LIN {X 0,Y 254.644,Z 265.777,A -85,B 0,C 180,E1 -18845.153,E2 -18845.153} C_VEL
LIN {X 0,Y 252.465,Z 261.449,A -85,B 0,C 180,E1 -18845.727,E2 -18845.727} C_VEL
LIN {X 0,Y 250.653,Z 254.367,A -85,B 0,C 180,E1 -18848.916,E2 -18848.916} C_VEL
LIN {X 0,Y 249.032,Z 248.465,A -85,B 0,C 180,E1 -18851.812,E2 -18851.812} C_VEL
LIN {X 0,Y 248.993,Z 248.471,A -85,B 0,C 180,E1 -18855.118,E2 -18855.118} C_VEL
LIN {X 0,Y 248.985,Z 248.471,A -85,B 0,C 180,E1 -18859.518,E2 -18859.518} C_VEL
LIN {X 0,Y 249.027,Z 248.458,A -85,B 0,C 180,E1 -18863.654,E2 -18863.654} C_VEL
LIN {X 0,Y 249.034,Z 248.461,A -85,B 0,C 180,E1 -18867.847,E2 -18867.847} C_VEL
LIN {X 0,Y 249.054,Z 248.454,A -85,B 0,C 180,E1 -18871.333,E2 -18871.333} C_VEL
LIN {X 0,Y 249.125,Z 248.443,A -85,B 0,C 180,E1 -18874.966,E2 -18874.966} C_VEL
LIN {X 0,Y 249.09,Z 248.448,A -85,B 0,C 180,E1 -18878.605,E2 -18878.605} C_VEL
LIN {X 0,Y 249.196,Z 248.434,A -85,B 0,C 180,E1 -18883.619,E2 -18883.619} C_VEL
LIN {X 0,Y 249.253,Z 248.426,A -85,B 0,C 180,E1 -18888.617,E2 -18888.617} C_VEL
LIN {X 0,Y 249.481,Z 248.4,A -85,B 0,C 180,E1 -18891.903,E2 -18891.903} C_VEL
LIN {X 0,Y 249.424,Z 248.409,A -85,B 0,C 180,E1 -18896.77,E2 -18896.77} C_VEL
LIN {X 0,Y 249.722,Z 248.378,A -85,B 0,C 180,E1 -18900,E2 -18900} C_VEL
LIN {X 0,Y 249.428,Z 248.403,A -85,B 0,C 180,E1 -18903.231,E2 -18903.231} C_VEL
LIN {X 0,Y 249.428,Z 248.412,A -85,B 0,C 180,E1 -18906.539,E2 -18906.539} C_VEL
LIN {X 0,Y 249.344,Z 248.42,A -85,B 0,C 180,E1 -18909.737,E2 -18909.737} C_VEL
LIN {X 0,Y 249.184,Z 248.44,A -85,B 0,C 180,E1 -18914.705,E2 -18914.705} C_VEL
LIN {X 0,Y 249.122,Z 248.44,A -85,B 0,C 180,E1 -18918.079,E2 -18918.079} C_VEL
LIN {X 0,Y 249.089,Z 248.449,A -85,B 0,C 180,E1 -18921.518,E2 -18921.518} C_VEL
LIN {X 0,Y 249.132,Z 248.446,A -85,B 0,C 180,E1 -18925.482,E2 -18925.482} C_VEL
LIN {X 0,Y 249.084,Z 248.456,A -85,B 0,C 180,E1 -18928.993,E2 -18928.993} C_VEL
LIN {X 0,Y 249.038,Z 248.463,A -85,B 0,C 180,E1 -18932.425,E2 -18932.425} C_VEL
LIN {X 0,Y 249.071,Z 248.454,A -85,B 0,C 180,E1 -18936.339,E2 -18936.339} C_VEL
LIN {X 0,Y 249.028,Z 248.466,A -85,B 0,C 180,E1 -18940.474,E2 -18940.474} C_VEL
LIN {X 0,Y 249.009,Z 248.471,A -85,B 0,C 180,E1 -18944.878,E2 -18944.878} C_VEL
LIN {X 0,Y 249.053,Z 248.62,A -85,B 0,C 180,E1 -18946.775,E2 -18946.775} C_VEL
LIN {X 0,Y 249.732,Z 251.001,A -85,B 0,C 180,E1 -18947.867,E2 -18947.867} C_VEL
LIN {X 0,Y 251.958,Z 254.871,A -85,B 0,C 180,E1 -18948.414,E2 -18948.414} C_VEL
LIN {X 0,Y 259.682,Z 268.72,A -85,B 0,C 180,E1 -18950.225,E2 -18950.225} C_VEL
LIN {X 0,Y 266.813,Z 283.218,A -85,B 0,C 180,E1 -18951.823,E2 -18951.823} C_VEL
LIN {X 0,Y 272.007,Z 295.388,A -85,B 0,C 180,E1 -18952.966,E2 -18952.966} C_VEL
LIN {X 0,Y 269.432,Z 358.338,A -85,B 0,C 180,E1 -18954.619,E2 -18954.619} C_VEL
LIN {X 0,Y 268.302,Z 371.737,A -85,B 0,C 180,E1 -18955.269,E2 -18955.269} C_VEL
LIN {X 0,Y 266.695,Z 384.328,A -85,B 0,C 180,E1 -18956.173,E2 -18956.173} C_VEL
LIN {X 0,Y 264.837,Z 395.51,A -85,B 0,C 180,E1 -18957.269,E2 -18957.269} C_VEL
LIN {X 0,Y 262.78,Z 405.83,A -85,B 0,C 180,E1 -18958.566,E2 -18958.566} C_VEL
LIN {X 0,Y 260.538,Z 415.694,A -85,B 0,C 180,E1 -18960.123,E2 -18960.123} C_VEL
LIN {X 0,Y 257.968,Z 425.167,A -85,B 0,C 180,E1 -18961.969,E2 -18961.969} C_VEL
LIN {X 0,Y 255.795,Z 433.148,A -85,B 0,C 180,E1 -18963.921,E2 -18963.921} C_VEL
LIN {X 0,Y 253.647,Z 440.407,A -85,B 0,C 180,E1 -18966.115,E2 -18966.115} C_VEL
LIN {X 0,Y 251.531,Z 447.119,A -85,B 0,C 180,E1 -18968.701,E2 -18968.701} C_VEL
LIN {X 0,Y 249.932,Z 452.023,A -85,B 0,C 180,E1 -18971.133,E2 -18971.133} C_VEL
LIN {X 0,Y 248.6,Z 456.301,A -85,B 0,C 180,E1 -18973.987,E2 -18973.987} C_VEL
LIN {X 0,Y 247.593,Z 459.227,A -85,B 0,C 180,E1 -18976.875,E2 -18976.875} C_VEL
LIN {X 0,Y 246.978,Z 460.932,A -85,B 0,C 180,E1 -18980.169,E2 -18980.169} C_VEL
LIN {X 0,Y 246.875,Z 461.202,A -85,B 0,C 180,E1 -18981.817,E2 -18981.817} C_VEL
LIN {X 0,Y 246.896,Z 461.079,A -85,B 0,C 180,E1 -18983.462,E2 -18983.462} C_VEL
LIN {X 0,Y 246.904,Z 460.527,A -85,B 0,C 180,E1 -18985.101,E2 -18985.101} C_VEL
LIN {X 0,Y 246.944,Z 459.589,A -85,B 0,C 180,E1 -18986.737,E2 -18986.737} C_VEL
LIN {X 0,Y 247.065,Z 458.263,A -85,B 0,C 180,E1 -18988.37,E2 -18988.37} C_VEL
LIN {X 0,Y 247.333,Z 455.467,A -85,B 0,C 180,E1 -18990.814,E2 -18990.814} C_VEL
LIN {X 0,Y 247.846,Z 451.66,A -85,B 0,C 180,E1 -18993.251,E2 -18993.251} C_VEL
LIN {X 0,Y 248.73,Z 446.732,A -85,B 0,C 180,E1 -18995.675,E2 -18995.675} C_VEL
LIN {X 0,Y 249.83,Z 440.548,A -85,B 0,C 180,E1 -18998.086,E2 -18998.086} C_VEL
LIN {X 0,Y 251.372,Z 432.816,A -85,B 0,C 180,E1 -19000.471,E2 -19000.471} C_VEL
LIN {X 0,Y 253.2,Z 423.156,A -85,B 0,C 180,E1 -19002.83,E2 -19002.83} C_VEL
LIN {X 0,Y 255.034,Z 413.156,A -85,B 0,C 180,E1 -19004.768,E2 -19004.768} C_VEL
LIN {X 0,Y 256.708,Z 402.883,A -85,B 0,C 180,E1 -19006.349,E2 -19006.349} C_VEL
LIN {X 0,Y 258.418,Z 390.457,A -85,B 0,C 180,E1 -19007.847,E2 -19007.847} C_VEL
LIN {X 0,Y 259.785,Z 378.325,A -85,B 0,C 180,E1 -19008.944,E2 -19008.944} C_VEL
LIN {X 0,Y 260.762,Z 365.091,A -85,B 0,C 180,E1 -19009.79,E2 -19009.79} C_VEL
LIN {X 0,Y 261.46,Z 352.137,A -85,B 0,C 180,E1 -19010.299,E2 -19010.299} C_VEL
LIN {X 0,Y 263.463,Z 286.138,A -85,B 0,C 180,E1 -19012.052,E2 -19012.052} C_VEL
LIN {X 0,Y 262.345,Z 281.579,A -85,B 0,C 180,E1 -19012.305,E2 -19012.305} C_VEL
LIN {X 0,Y 255.624,Z 264.114,A -85,B 0,C 180,E1 -19013.578,E2 -19013.578} C_VEL
LIN {X 0,Y 249.495,Z 250.179,A -85,B 0,C 180,E1 -19014.754,E2 -19014.754} C_VEL
LIN {X 0,Y 249.1,Z 248.457,A -85,B 0,C 180,E1 -19015.573,E2 -19015.573} C_VEL
LIN {X 0,Y 249.043,Z 248.465,A -85,B 0,C 180,E1 -19018.976,E2 -19018.976} C_VEL
LIN {X 0,Y 249.029,Z 248.466,A -85,B 0,C 180,E1 -19022.426,E2 -19022.426} C_VEL
LIN {X 0,Y 249.05,Z 248.462,A -85,B 0,C 180,E1 -19026.342,E2 -19026.342} C_VEL
LIN {X 0,Y 249.008,Z 248.467,A -85,B 0,C 180,E1 -19030.478,E2 -19030.478} C_VEL
LIN {X 0,Y 249.009,Z 248.468,A -85,B 0,C 180,E1 -19034.878,E2 -19034.878} C_VEL
LIN {X 0,Y 249.02,Z 248.464,A -85,B 0,C 180,E1 -19037.363,E2 -19037.363} C_VEL
LIN {X 0,Y 249.045,Z 248.46,A -85,B 0,C 180,E1 -19042.2,E2 -19042.2} C_VEL
LIN {X 0,Y 249.045,Z 248.456,A -85,B 0,C 180,E1 -19045.639,E2 -19045.639} C_VEL
LIN {X 0,Y 249.048,Z 248.454,A -85,B 0,C 180,E1 -19049.472,E2 -19049.472} C_VEL
LIN {X 0,Y 249.073,Z 248.457,A -85,B 0,C 180,E1 -19053.162,E2 -19053.162} C_VEL
LIN {X 0,Y 249.08,Z 248.438,A -85,B 0,C 180,E1 -19056.732,E2 -19056.732} C_VEL
LIN {X 0,Y 249.112,Z 248.443,A -85,B 0,C 180,E1 -19060.211,E2 -19060.211} C_VEL
LIN {X 0,Y 249.243,Z 248.434,A -85,B 0,C 180,E1 -19063.622,E2 -19063.622} C_VEL
LIN {X 0,Y 249.244,Z 248.412,A -85,B 0,C 180,E1 -19068.616,E2 -19068.616} C_VEL
LIN {X 0,Y 249.42,Z 248.405,A -85,B 0,C 180,E1 -19071.901,E2 -19071.901} C_VEL
LIN {X 0,Y 249.286,Z 248.43,A -85,B 0,C 180,E1 -19075.148,E2 -19075.148} C_VEL
LIN {X 0,Y 249.675,Z 248.377,A -85,B 0,C 180,E1 -19078.387,E2 -19078.387} C_VEL
LIN {X 0,Y 249.675,Z 248.381,A -85,B 0,C 180,E1 -19081.613,E2 -19081.613} C_VEL
LIN {X 0,Y 249.374,Z 248.413,A -85,B 0,C 180,E1 -19083.673,E2 -19083.673} C_VEL
LIN {X 0,Y 248.627,Z 248.513,A -85,B 0,C 180,E1 -19085.022,E2 -19085.022} C_VEL
LIN {X 0,Y 245.805,Z 248.865,A -85,B 0,C 180,E1 -19087.226,E2 -19087.226} C_VEL
LIN {X 0,Y 242.607,Z 249.259,A -85,B 0,C 180,E1 -19089.94,E2 -19089.94} C_VEL
LIN {X 0,Y 242.238,Z 249.299,A -85,B 0,C 180,E1 -19090.879,E2 -19090.879} C_VEL
LIN {X 0,Y 242.127,Z 249.323,A -85,B 0,C 180,E1 -19095.143,E2 -19095.143} C_VEL
LIN {X 0,Y 242.042,Z 249.326,A -85,B 0,C 180,E1 -19098.626,E2 -19098.626} C_VEL
LIN {X 0,Y 242.003,Z 249.34,A -85,B 0,C 180,E1 -19102.181,E2 -19102.181} C_VEL
LIN {X 0,Y 242.032,Z 249.33,A -85,B 0,C 180,E1 -19105.821,E2 -19105.821} C_VEL
LIN {X 0,Y 241.97,Z 249.34,A -85,B 0,C 180,E1 -19109.588,E2 -19109.588} C_VEL
LIN {X 0,Y 241.979,Z 249.341,A -85,B 0,C 180,E1 -19113.493,E2 -19113.493} C_VEL
LIN {X 0,Y 241.987,Z 249.34,A -85,B 0,C 180,E1 -19117.582,E2 -19117.582} C_VEL
LIN {X 0,Y 241.923,Z 249.348,A -85,B 0,C 180,E1 -19121.925,E2 -19121.925} C_VEL
LIN {X 0,Y 241.932,Z 249.348,A -85,B 0,C 180,E1 -19126.572,E2 -19126.572} C_VEL
LIN {X 0,Y 241.958,Z 249.344,A -85,B 0,C 180,E1 -19130.281,E2 -19130.281} C_VEL
LIN {X 0,Y 242.041,Z 249.382,A -85,B 0,C 180,E1 -19133.562,E2 -19133.562} C_VEL
LIN {X 0,Y 243.819,Z 257.168,A -85,B 0,C 180,E1 -19136.793,E2 -19136.793} C_VEL
LIN {X 0,Y 244.838,Z 261.978,A -85,B 0,C 180,E1 -19138.697,E2 -19138.697} C_VEL
LIN {X 0,Y 252.327,Z 280.988,A -85,B 0,C 180,E1 -19140.214,E2 -19140.214} C_VEL
LIN {X 0,Y 256.148,Z 308.906,A -85,B 0,C 180,E1 -19141.504,E2 -19141.504} C_VEL
LIN {X 0,Y 256.345,Z 314.755,A -85,B 0,C 180,E1 -19141.703,E2 -19141.703} C_VEL
LIN {X 0,Y 254.429,Z 371.318,A -85,B 0,C 180,E1 -19143.279,E2 -19143.279} C_VEL
LIN {X 0,Y 253.423,Z 384.264,A -85,B 0,C 180,E1 -19143.936,E2 -19143.936} C_VEL
LIN {X 0,Y 252.068,Z 396.315,A -85,B 0,C 180,E1 -19144.837,E2 -19144.837} C_VEL
LIN {X 0,Y 250.514,Z 407.691,A -85,B 0,C 180,E1 -19145.997,E2 -19145.997} C_VEL
LIN {X 0,Y 248.618,Z 419.413,A -85,B 0,C 180,E1 -19147.566,E2 -19147.566} C_VEL
LIN {X 0,Y 246.636,Z 429.94,A -85,B 0,C 180,E1 -19149.352,E2 -19149.352} C_VEL
LIN {X 0,Y 244.93,Z 439.63,A -85,B 0,C 180,E1 -19151.437,E2 -19151.437} C_VEL
LIN {X 0,Y 243.337,Z 447.877,A -85,B 0,C 180,E1 -19153.644,E2 -19153.644} C_VEL
LIN {X 0,Y 241.887,Z 455.347,A -85,B 0,C 180,E1 -19156.131,E2 -19156.131} C_VEL
LIN {X 0,Y 240.786,Z 462.227,A -85,B 0,C 180,E1 -19159.064,E2 -19159.064} C_VEL
LIN {X 0,Y 240.201,Z 466.755,A -85,B 0,C 180,E1 -19161.588,E2 -19161.588} C_VEL
LIN {X 0,Y 239.958,Z 469.138,A -85,B 0,C 180,E1 -19163.272,E2 -19163.272} C_VEL
LIN {X 0,Y 239.795,Z 471.343,A -85,B 0,C 180,E1 -19165.196,E2 -19165.196} C_VEL
LIN {X 0,Y 239.841,Z 473.685,A -85,B 0,C 180,E1 -19168.321,E2 -19168.321} C_VEL
LIN {X 0,Y 239.913,Z 474.357,A -85,B 0,C 180,E1 -19170,E2 -19170} C_VEL
LIN {X 0,Y 239.831,Z 474.635,A -85,B 0,C 180,E1 -19171.679,E2 -19171.679} C_VEL
LIN {X 0,Y 239.791,Z 474.103,A -85,B 0,C 180,E1 -19174.794,E2 -19174.794} C_VEL
LIN {X 0,Y 239.956,Z 473.052,A -85,B 0,C 180,E1 -19176.728,E2 -19176.728} C_VEL
LIN {X 0,Y 240.683,Z 470,A -85,B 0,C 180,E1 -19180.09,E2 -19180.09} C_VEL
LIN {X 0,Y 241.64,Z 466.547,A -85,B 0,C 180,E1 -19182.6,E2 -19182.6} C_VEL
LIN {X 0,Y 243.009,Z 462.026,A -85,B 0,C 180,E1 -19185.087,E2 -19185.087} C_VEL
LIN {X 0,Y 245.254,Z 455.196,A -85,B 0,C 180,E1 -19187.942,E2 -19187.942} C_VEL
LIN {X 0,Y 247.765,Z 446.972,A -85,B 0,C 180,E1 -19190.599,E2 -19190.599} C_VEL
LIN {X 0,Y 250.142,Z 438.63,A -85,B 0,C 180,E1 -19192.726,E2 -19192.726} C_VEL
LIN {X 0,Y 253.127,Z 428.044,A -85,B 0,C 180,E1 -19194.831,E2 -19194.831} C_VEL
LIN {X 0,Y 255.775,Z 417.28,A -85,B 0,C 180,E1 -19196.52,E2 -19196.52} C_VEL
LIN {X 0,Y 258.067,Z 406.797,A -85,B 0,C 180,E1 -19197.799,E2 -19197.799} C_VEL
LIN {X 0,Y 260.336,Z 394.187,A -85,B 0,C 180,E1 -19198.963,E2 -19198.963} C_VEL
LIN {X 0,Y 261.944,Z 381.626,A -85,B 0,C 180,E1 -19199.815,E2 -19199.815} C_VEL
LIN {X 0,Y 263.192,Z 368.388,A -85,B 0,C 180,E1 -19200.377,E2 -19200.377} C_VEL
LIN {X 0,Y 265.289,Z 315.913,A -85,B 0,C 180,E1 -19201.779,E2 -19201.779} C_VEL
LIN {X 0,Y 262.4,Z 297.114,A -85,B 0,C 180,E1 -19202.824,E2 -19202.824} C_VEL
LIN {X 0,Y 256.064,Z 282.546,A -85,B 0,C 180,E1 -19204.33,E2 -19204.33} C_VEL
LIN {X 0,Y 249.272,Z 269.095,A -85,B 0,C 180,E1 -19205.99,E2 -19205.99} C_VEL
LIN {X 0,Y 246.784,Z 264.532,A -85,B 0,C 180,E1 -19206.617,E2 -19206.617} C_VEL
LIN {X 0,Y 245.247,Z 261.249,A -85,B 0,C 180,E1 -19207.051,E2 -19207.051} C_VEL
LIN {X 0,Y 242.861,Z 252.644,A -85,B 0,C 180,E1 -19211.201,E2 -19211.201} C_VEL
LIN {X 0,Y 241.974,Z 249.345,A -85,B 0,C 180,E1 -19212.993,E2 -19212.993} C_VEL
LIN {X 0,Y 241.923,Z 249.351,A -85,B 0,C 180,E1 -19216.574,E2 -19216.574} C_VEL
LIN {X 0,Y 241.992,Z 249.341,A -85,B 0,C 180,E1 -19221.641,E2 -19221.641} C_VEL
LIN {X 0,Y 241.98,Z 249.341,A -85,B 0,C 180,E1 -19224.488,E2 -19224.488} C_VEL
LIN {X 0,Y 241.954,Z 249.345,A -85,B 0,C 180,E1 -19228.477,E2 -19228.477} C_VEL
LIN {X 0,Y 241.973,Z 249.343,A -85,B 0,C 180,E1 -19232.308,E2 -19232.308} C_VEL
LIN {X 0,Y 242.035,Z 249.335,A -85,B 0,C 180,E1 -19236.014,E2 -19236.014} C_VEL
LIN {X 0,Y 242.022,Z 249.33,A -85,B 0,C 180,E1 -19239.607,E2 -19239.607} C_VEL
LIN {X 0,Y 242.116,Z 249.316,A -85,B 0,C 180,E1 -19243.316,E2 -19243.316} C_VEL
LIN {X 0,Y 242.185,Z 249.305,A -85,B 0,C 180,E1 -19248.28,E2 -19248.28} C_VEL
LIN {X 0,Y 242.428,Z 249.28,A -85,B 0,C 180,E1 -19251.666,E2 -19251.666} C_VEL
LIN {X 0,Y 242.248,Z 249.306,A -85,B 0,C 180,E1 -19255.007,E2 -19255.007} C_VEL
LIN {X 0,Y 242.632,Z 249.248,A -85,B 0,C 180,E1 -19258.34,E2 -19258.34} C_VEL
LIN {X 0,Y 242.634,Z 249.256,A -85,B 0,C 180,E1 -19261.66,E2 -19261.66} C_VEL
LIN {X 0,Y 242.402,Z 249.289,A -85,B 0,C 180,E1 -19266.66,E2 -19266.66} C_VEL
LIN {X 0,Y 242.267,Z 249.305,A -85,B 0,C 180,E1 -19270.024,E2 -19270.024} C_VEL
LIN {X 0,Y 242.14,Z 249.319,A -85,B 0,C 180,E1 -19275.143,E2 -19275.143} C_VEL
LIN {X 0,Y 242.062,Z 249.32,A -85,B 0,C 180,E1 -19278.625,E2 -19278.625} C_VEL
LIN {X 0,Y 242.014,Z 249.326,A -85,B 0,C 180,E1 -19282.18,E2 -19282.18} C_VEL
LIN {X 0,Y 242.068,Z 249.323,A -85,B 0,C 180,E1 -19285.838,E2 -19285.838} C_VEL
LIN {X 0,Y 242.032,Z 249.33,A -85,B 0,C 180,E1 -19289.58,E2 -19289.58} C_VEL
LIN {X 0,Y 241.993,Z 249.336,A -85,B 0,C 180,E1 -19293.491,E2 -19293.491} C_VEL
LIN {X 0,Y 242.004,Z 249.341,A -85,B 0,C 180,E1 -19297.58,E2 -19297.58} C_VEL
LIN {X 0,Y 241.946,Z 249.345,A -85,B 0,C 180,E1 -19301.921,E2 -19301.921} C_VEL
LIN {X 0,Y 241.989,Z 249.526,A -85,B 0,C 180,E1 -19305.666,E2 -19305.666} C_VEL
LIN {X 0,Y 242.518,Z 251.239,A -85,B 0,C 180,E1 -19306.48,E2 -19306.48} C_VEL
LIN {X 0,Y 244.824,Z 255.198,A -85,B 0,C 180,E1 -19307.087,E2 -19307.087} C_VEL
LIN {X 0,Y 252.458,Z 268.434,A -85,B 0,C 180,E1 -19308.985,E2 -19308.985} C_VEL
LIN {X 0,Y 259.973,Z 283.303,A -85,B 0,C 180,E1 -19310.763,E2 -19310.763} C_VEL
LIN {X 0,Y 266.007,Z 297.202,A -85,B 0,C 180,E1 -19312.153,E2 -19312.153} C_VEL
LIN {X 0,Y 263.489,Z 358.084,A -85,B 0,C 180,E1 -19313.784,E2 -19313.784} C_VEL
LIN {X 0,Y 262.384,Z 371.255,A -85,B 0,C 180,E1 -19314.427,E2 -19314.427} C_VEL
LIN {X 0,Y 260.789,Z 383.471,A -85,B 0,C 180,E1 -19315.299,E2 -19315.299} C_VEL
LIN {X 0,Y 258.862,Z 394.95,A -85,B 0,C 180,E1 -19316.415,E2 -19316.415} C_VEL
LIN {X 0,Y 256.658,Z 405.402,A -85,B 0,C 180,E1 -19317.726,E2 -19317.726} C_VEL
LIN {X 0,Y 254.213,Z 415.793,A -85,B 0,C 180,E1 -19319.389,E2 -19319.389} C_VEL
LIN {X 0,Y 251.641,Z 424.936,A -85,B 0,C 180,E1 -19321.199,E2 -19321.199} C_VEL
LIN {X 0,Y 249.326,Z 432.987,A -85,B 0,C 180,E1 -19323.192,E2 -19323.192} C_VEL
LIN {X 0,Y 246.916,Z 440.834,A -85,B 0,C 180,E1 -19325.62,E2 -19325.62} C_VEL
LIN {X 0,Y 244.835,Z 447.097,A -85,B 0,C 180,E1 -19328.089,E2 -19328.089} C_VEL
LIN {X 0,Y 243.12,Z 452.049,A -85,B 0,C 180,E1 -19330.583,E2 -19330.583} C_VEL
LIN {X 0,Y 241.866,Z 455.855,A -85,B 0,C 180,E1 -19333.108,E2 -19333.108} C_VEL
LIN {X 0,Y 241.182,Z 457.808,A -85,B 0,C 180,E1 -19334.796,E2 -19334.796} C_VEL
LIN {X 0,Y 240.616,Z 459.344,A -85,B 0,C 180,E1 -19336.487,E2 -19336.487} C_VEL
LIN {X 0,Y 240.153,Z 460.428,A -85,B 0,C 180,E1 -19338.179,E2 -19338.179} C_VEL
LIN {X 0,Y 239.798,Z 461.39,A -85,B 0,C 180,E1 -19341.573,E2 -19341.573} C_VEL
LIN {X 0,Y 239.788,Z 461.294,A -85,B 0,C 180,E1 -19343.267,E2 -19343.267} C_VEL
LIN {X 0,Y 239.804,Z 460.669,A -85,B 0,C 180,E1 -19345.173,E2 -19345.173} C_VEL
LIN {X 0,Y 239.966,Z 458.546,A -85,B 0,C 180,E1 -19348.322,E2 -19348.322} C_VEL
LIN {X 0,Y 240.248,Z 455.79,A -85,B 0,C 180,E1 -19350.838,E2 -19350.838} C_VEL
LIN {X 0,Y 240.771,Z 452.026,A -85,B 0,C 180,E1 -19353.347,E2 -19353.347} C_VEL
LIN {X 0,Y 241.675,Z 447.145,A -85,B 0,C 180,E1 -19355.842,E2 -19355.842} C_VEL
LIN {X 0,Y 242.82,Z 441.011,A -85,B 0,C 180,E1 -19358.321,E2 -19358.321} C_VEL
LIN {X 0,Y 244.417,Z 433.366,A -85,B 0,C 180,E1 -19360.772,E2 -19360.772} C_VEL
LIN {X 0,Y 246.316,Z 423.776,A -85,B 0,C 180,E1 -19363.195,E2 -19363.195} C_VEL
LIN {X 0,Y 248.217,Z 413.88,A -85,B 0,C 180,E1 -19365.183,E2 -19365.183} C_VEL
LIN {X 0,Y 250.058,Z 403.078,A -85,B 0,C 180,E1 -19366.897,E2 -19366.897} C_VEL
LIN {X 0,Y 251.639,Z 392.119,A -85,B 0,C 180,E1 -19368.27,E2 -19368.27} C_VEL
LIN {X 0,Y 253.115,Z 379.659,A -85,B 0,C 180,E1 -19369.463,E2 -19369.463} C_VEL
LIN {X 0,Y 254.184,Z 367.02,A -85,B 0,C 180,E1 -19370.325,E2 -19370.325} C_VEL
LIN {X 0,Y 254.817,Z 355.22,A -85,B 0,C 180,E1 -19370.852,E2 -19370.852} C_VEL
LIN {X 0,Y 257.05,Z 287.162,A -85,B 0,C 180,E1 -19372.709,E2 -19372.709} C_VEL
LIN {X 0,Y 255.55,Z 282.213,A -85,B 0,C 180,E1 -19373.027,E2 -19373.027} C_VEL
LIN {X 0,Y 249.926,Z 267.53,A -85,B 0,C 180,E1 -19374.141,E2 -19374.141} C_VEL
LIN {X 0,Y 242.234,Z 250.331,A -85,B 0,C 180,E1 -19375.704,E2 -19375.704} C_VEL
LIN {X 0,Y 242.011,Z 249.341,A -85,B 0,C 180,E1 -19376.24,E2 -19376.24} C_VEL
LIN {X 0,Y 241.972,Z 249.343,A -85,B 0,C 180,E1 -19379.588,E2 -19379.588} C_VEL
LIN {X 0,Y 241.981,Z 249.342,A -85,B 0,C 180,E1 -19383.492,E2 -19383.492} C_VEL
LIN {X 0,Y 241.991,Z 249.34,A -85,B 0,C 180,E1 -19387.581,E2 -19387.581} C_VEL
LIN {X 0,Y 241.94,Z 249.345,A -85,B 0,C 180,E1 -19391.922,E2 -19391.922} C_VEL
LIN {X 0,Y 241.938,Z 249.349,A -85,B 0,C 180,E1 -19396.57,E2 -19396.57} C_VEL
LIN {X 0,Y 241.958,Z 249.346,A -85,B 0,C 180,E1 -19400.281,E2 -19400.281} C_VEL
LIN {X 0,Y 241.989,Z 249.341,A -85,B 0,C 180,E1 -19404.489,E2 -19404.489} C_VEL
LIN {X 0,Y 241.974,Z 249.325,A -85,B 0,C 180,E1 -19408.479,E2 -19408.479} C_VEL
LIN {X 0,Y 242.004,Z 249.339,A -85,B 0,C 180,E1 -19412.312,E2 -19412.312} C_VEL
LIN {X 0,Y 242.058,Z 249.319,A -85,B 0,C 180,E1 -19416.016,E2 -19416.016} C_VEL
LIN {X 0,Y 242.039,Z 249.322,A -85,B 0,C 180,E1 -19419.608,E2 -19419.608} C_VEL
LIN {X 0,Y 242.164,Z 249.316,A -85,B 0,C 180,E1 -19423.278,E2 -19423.278} C_VEL
LIN {X 0,Y 242.181,Z 249.292,A -85,B 0,C 180,E1 -19428.279,E2 -19428.279} C_VEL
LIN {X 0,Y 242.373,Z 249.282,A -85,B 0,C 180,E1 -19431.663,E2 -19431.663} C_VEL
LIN {X 0,Y 242.246,Z 249.307,A -85,B 0,C 180,E1 -19435.007,E2 -19435.007} C_VEL
LIN {X 0,Y 242.635,Z 249.253,A -85,B 0,C 180,E1 -19438.34,E2 -19438.34} C_VEL
LIN {X 0,Y 242.635,Z 249.258,A -85,B 0,C 180,E1 -19441.66,E2 -19441.66} C_VEL
LIN {X 0,Y 242.434,Z 249.288,A -85,B 0,C 180,E1 -19446.659,E2 -19446.659} C_VEL
LIN {X 0,Y 242.346,Z 249.291,A -85,B 0,C 180,E1 -19450.02,E2 -19450.02} C_VEL
LIN {X 0,Y 242.238,Z 249.299,A -85,B 0,C 180,E1 -19450.879,E2 -19450.879} C_VEL
LIN {X 0,Y 241.474,Z 249.397,A -85,B 0,C 180,E1 -19452.266,E2 -19452.266} C_VEL
LIN {X 0,Y 238.548,Z 249.771,A -85,B 0,C 180,E1 -19454.528,E2 -19454.528} C_VEL
LIN {X 0,Y 236.108,Z 250.073,A -85,B 0,C 180,E1 -19456.371,E2 -19456.371} C_VEL
LIN {X 0,Y 235.061,Z 250.197,A -85,B 0,C 180,E1 -19457.802,E2 -19457.802} C_VEL
LIN {X 0,Y 234.971,Z 250.205,A -85,B 0,C 180,E1 -19458.287,E2 -19458.287} C_VEL
LIN {X 0,Y 234.986,Z 250.213,A -85,B 0,C 180,E1 -19462.005,E2 -19462.005} C_VEL
LIN {X 0,Y 234.946,Z 250.217,A -85,B 0,C 180,E1 -19466.66,E2 -19466.66} C_VEL
LIN {X 0,Y 234.899,Z 250.22,A -85,B 0,C 180,E1 -19470.572,E2 -19470.572} C_VEL
LIN {X 0,Y 234.93,Z 250.217,A -85,B 0,C 180,E1 -19474.638,E2 -19474.638} C_VEL
LIN {X 0,Y 234.911,Z 250.22,A -85,B 0,C 180,E1 -19478.935,E2 -19478.935} C_VEL
LIN {X 0,Y 234.876,Z 250.227,A -85,B 0,C 180,E1 -19483.489,E2 -19483.489} C_VEL
LIN {X 0,Y 234.885,Z 250.226,A -85,B 0,C 180,E1 -19486.514,E2 -19486.514} C_VEL
LIN {X 0,Y 234.922,Z 250.22,A -85,B 0,C 180,E1 -19491.079,E2 -19491.079} C_VEL
LIN {X 0,Y 234.991,Z 250.273,A -85,B 0,C 180,E1 -19492.861,E2 -19492.861} C_VEL
LIN {X 0,Y 237.052,Z 259.31,A -85,B 0,C 180,E1 -19496.738,E2 -19496.738} C_VEL
LIN {X 0,Y 237.647,Z 261.991,A -85,B 0,C 180,E1 -19497.753,E2 -19497.753} C_VEL
LIN {X 0,Y 244.944,Z 279.897,A -85,B 0,C 180,E1 -19499.295,E2 -19499.295} C_VEL
LIN {X 0,Y 246.394,Z 284.268,A -85,B 0,C 180,E1 -19499.615,E2 -19499.615} C_VEL
LIN {X 0,Y 249.991,Z 311.683,A -85,B 0,C 180,E1 -19500.91,E2 -19500.91} C_VEL
LIN {X 0,Y 247.972,Z 371.131,A -85,B 0,C 180,E1 -19502.609,E2 -19502.609} C_VEL
LIN {X 0,Y 246.883,Z 384.479,A -85,B 0,C 180,E1 -19503.305,E2 -19503.305} C_VEL
LIN {X 0,Y 245.4,Z 397.49,A -85,B 0,C 180,E1 -19504.331,E2 -19504.331} C_VEL
LIN {X 0,Y 243.497,Z 410.101,A -85,B 0,C 180,E1 -19505.714,E2 -19505.714} C_VEL
LIN {X 0,Y 241.552,Z 421.344,A -85,B 0,C 180,E1 -19507.325,E2 -19507.325} C_VEL
LIN {X 0,Y 239.755,Z 430.429,A -85,B 0,C 180,E1 -19508.956,E2 -19508.956} C_VEL
LIN {X 0,Y 238.016,Z 439.757,A -85,B 0,C 180,E1 -19511.047,E2 -19511.047} C_VEL
LIN {X 0,Y 236.482,Z 447.434,A -85,B 0,C 180,E1 -19513.157,E2 -19513.157} C_VEL
LIN {X 0,Y 234.978,Z 454.949,A -85,B 0,C 180,E1 -19515.715,E2 -19515.715} C_VEL
LIN {X 0,Y 233.775,Z 461.881,A -85,B 0,C 180,E1 -19518.731,E2 -19518.731} C_VEL
LIN {X 0,Y 233.142,Z 466.445,A -85,B 0,C 180,E1 -19521.331,E2 -19521.331} C_VEL
LIN {X 0,Y 232.891,Z 468.845,A -85,B 0,C 180,E1 -19523.067,E2 -19523.067} C_VEL
LIN {X 0,Y 232.714,Z 471.294,A -85,B 0,C 180,E1 -19525.278,E2 -19525.278} C_VEL
LIN {X 0,Y 232.752,Z 473.453,A -85,B 0,C 180,E1 -19528.27,E2 -19528.27} C_VEL
LIN {X 0,Y 232.823,Z 474.139,A -85,B 0,C 180,E1 -19530,E2 -19530} C_VEL
LIN {X 0,Y 232.743,Z 474.431,A -85,B 0,C 180,E1 -19531.73,E2 -19531.73} C_VEL
LIN {X 0,Y 232.707,Z 474.006,A -85,B 0,C 180,E1 -19534.702,E2 -19534.702} C_VEL
LIN {X 0,Y 232.894,Z 472.905,A -85,B 0,C 180,E1 -19536.933,E2 -19536.933} C_VEL
LIN {X 0,Y 233.681,Z 469.887,A -85,B 0,C 180,E1 -19540.396,E2 -19540.396} C_VEL
LIN {X 0,Y 234.672,Z 466.462,A -85,B 0,C 180,E1 -19542.98,E2 -19542.98} C_VEL
LIN {X 0,Y 236.157,Z 461.976,A -85,B 0,C 180,E1 -19545.536,E2 -19545.536} C_VEL
LIN {X 0,Y 238.474,Z 455.203,A -85,B 0,C 180,E1 -19548.47,E2 -19548.47} C_VEL
LIN {X 0,Y 240.92,Z 447.621,A -85,B 0,C 180,E1 -19551.015,E2 -19551.015} C_VEL
LIN {X 0,Y 243.601,Z 438.752,A -85,B 0,C 180,E1 -19553.372,E2 -19553.372} C_VEL
LIN {X 0,Y 246.727,Z 428.238,A -85,B 0,C 180,E1 -19555.521,E2 -19555.521} C_VEL
LIN {X 0,Y 249.454,Z 417.558,A -85,B 0,C 180,E1 -19557.247,E2 -19557.247} C_VEL
LIN {X 0,Y 251.835,Z 407.215,A -85,B 0,C 180,E1 -19558.549,E2 -19558.549} C_VEL
LIN {X 0,Y 254.18,Z 394.816,A -85,B 0,C 180,E1 -19559.734,E2 -19559.734} C_VEL
LIN {X 0,Y 255.931,Z 381.785,A -85,B 0,C 180,E1 -19560.646,E2 -19560.646} C_VEL
LIN {X 0,Y 257.233,Z 368.889,A -85,B 0,C 180,E1 -19561.215,E2 -19561.215} C_VEL
LIN {X 0,Y 259.356,Z 315.813,A -85,B 0,C 180,E1 -19562.677,E2 -19562.677} C_VEL
LIN {X 0,Y 256.73,Z 299.566,A -85,B 0,C 180,E1 -19563.639,E2 -19563.639} C_VEL
LIN {X 0,Y 250.701,Z 285.754,A -85,B 0,C 180,E1 -19565.138,E2 -19565.138} C_VEL
LIN {X 0,Y 244.162,Z 272.639,A -85,B 0,C 180,E1 -19566.816,E2 -19566.816} C_VEL
LIN {X 0,Y 239.939,Z 264.906,A -85,B 0,C 180,E1 -19567.944,E2 -19567.944} C_VEL
LIN {X 0,Y 237.882,Z 260.913,A -85,B 0,C 180,E1 -19568.571,E2 -19568.571} C_VEL
LIN {X 0,Y 235.596,Z 252.632,A -85,B 0,C 180,E1 -19572.801,E2 -19572.801} C_VEL
LIN {X 0,Y 234.903,Z 250.226,A -85,B 0,C 180,E1 -19574.196,E2 -19574.196} C_VEL
LIN {X 0,Y 234.865,Z 250.229,A -85,B 0,C 180,E1 -19578.828,E2 -19578.828} C_VEL
LIN {X 0,Y 234.918,Z 250.222,A -85,B 0,C 180,E1 -19581.079,E2 -19581.079} C_VEL
LIN {X 0,Y 234.926,Z 250.218,A -85,B 0,C 180,E1 -19585.361,E2 -19585.361} C_VEL
LIN {X 0,Y 234.9,Z 250.219,A -85,B 0,C 180,E1 -19589.428,E2 -19589.428} C_VEL
LIN {X 0,Y 234.97,Z 250.208,A -85,B 0,C 180,E1 -19593.806,E2 -19593.806} C_VEL
LIN {X 0,Y 234.991,Z 250.203,A -85,B 0,C 180,E1 -19598.968,E2 -19598.968} C_VEL
LIN {X 0,Y 235.057,Z 250.195,A -85,B 0,C 180,E1 -19603.092,E2 -19603.092} C_VEL
LIN {X 0,Y 235.116,Z 250.185,A -85,B 0,C 180,E1 -19607.922,E2 -19607.922} C_VEL
LIN {X 0,Y 235.377,Z 250.16,A -85,B 0,C 180,E1 -19611.414,E2 -19611.414} C_VEL
LIN {X 0,Y 235.403,Z 250.149,A -85,B 0,C 180,E1 -19613.141,E2 -19613.141} C_VEL
LIN {X 0,Y 235.592,Z 250.124,A -85,B 0,C 180,E1 -19618.291,E2 -19618.291} C_VEL
LIN {X 0,Y 235.594,Z 250.132,A -85,B 0,C 180,E1 -19621.71,E2 -19621.71} C_VEL
LIN {X 0,Y 235.353,Z 250.164,A -85,B 0,C 180,E1 -19626.86,E2 -19626.86} C_VEL
LIN {X 0,Y 235.213,Z 250.185,A -85,B 0,C 180,E1 -19630.328,E2 -19630.328} C_VEL
LIN {X 0,Y 235.095,Z 250.201,A -85,B 0,C 180,E1 -19635.608,E2 -19635.608} C_VEL
LIN {X 0,Y 235.002,Z 250.203,A -85,B 0,C 180,E1 -19639.206,E2 -19639.206} C_VEL
LIN {X 0,Y 234.963,Z 250.204,A -85,B 0,C 180,E1 -19642.883,E2 -19642.883} C_VEL
LIN {X 0,Y 234.971,Z 250.205,A -85,B 0,C 180,E1 -19646.657,E2 -19646.657} C_VEL
LIN {X 0,Y 234.934,Z 250.214,A -85,B 0,C 180,E1 -19650.568,E2 -19650.568} C_VEL
LIN {X 0,Y 234.962,Z 250.217,A -85,B 0,C 180,E1 -19654.633,E2 -19654.633} C_VEL
LIN {X 0,Y 234.943,Z 250.215,A -85,B 0,C 180,E1 -19658.945,E2 -19658.945} C_VEL
LIN {X 0,Y 234.892,Z 250.225,A -85,B 0,C 180,E1 -19663.485,E2 -19663.485} C_VEL
LIN {X 0,Y 234.921,Z 250.371,A -85,B 0,C 180,E1 -19664.434,E2 -19664.434} C_VEL
LIN {X 0,Y 235.231,Z 251.484,A -85,B 0,C 180,E1 -19664.96,E2 -19664.96} C_VEL
LIN {X 0,Y 236.986,Z 254.584,A -85,B 0,C 180,E1 -19665.464,E2 -19665.464} C_VEL
LIN {X 0,Y 238.679,Z 257.151,A -85,B 0,C 180,E1 -19665.922,E2 -19665.922} C_VEL
LIN {X 0,Y 246.235,Z 270.09,A -85,B 0,C 180,E1 -19667.91,E2 -19667.91} C_VEL
LIN {X 0,Y 253.137,Z 283.463,A -85,B 0,C 180,E1 -19669.632,E2 -19669.632} C_VEL
LIN {X 0,Y 259.557,Z 297.842,A -85,B 0,C 180,E1 -19671.183,E2 -19671.183} C_VEL
LIN {X 0,Y 260.183,Z 299.383,A -85,B 0,C 180,E1 -19671.333,E2 -19671.333} C_VEL
LIN {X 0,Y 257.512,Z 358.954,A -85,B 0,C 180,E1 -19672.956,E2 -19672.956} C_VEL
LIN {X 0,Y 256.311,Z 372.305,A -85,B 0,C 180,E1 -19673.633,E2 -19673.633} C_VEL
LIN {X 0,Y 254.576,Z 384.84,A -85,B 0,C 180,E1 -19674.568,E2 -19674.568} C_VEL
LIN {X 0,Y 252.577,Z 395.993,A -85,B 0,C 180,E1 -19675.705,E2 -19675.705} C_VEL
LIN {X 0,Y 250.317,Z 406.287,A -85,B 0,C 180,E1 -19677.045,E2 -19677.045} C_VEL
LIN {X 0,Y 247.955,Z 415.848,A -85,B 0,C 180,E1 -19678.611,E2 -19678.611} C_VEL
LIN {X 0,Y 245.376,Z 424.709,A -85,B 0,C 180,E1 -19680.391,E2 -19680.391} C_VEL
LIN {X 0,Y 242.909,Z 432.83,A -85,B 0,C 180,E1 -19682.424,E2 -19682.424} C_VEL
LIN {X 0,Y 240.434,Z 440.508,A -85,B 0,C 180,E1 -19684.82,E2 -19684.82} C_VEL
LIN {X 0,Y 238.173,Z 447.08,A -85,B 0,C 180,E1 -19687.443,E2 -19687.443} C_VEL
LIN {X 0,Y 236.349,Z 452.077,A -85,B 0,C 180,E1 -19690.004,E2 -19690.004} C_VEL
LIN {X 0,Y 234.985,Z 455.926,A -85,B 0,C 180,E1 -19692.597,E2 -19692.597} C_VEL
LIN {X 0,Y 234.259,Z 457.899,A -85,B 0,C 180,E1 -19694.335,E2 -19694.335} C_VEL
LIN {X 0,Y 233.637,Z 459.455,A -85,B 0,C 180,E1 -19696.075,E2 -19696.075} C_VEL
LIN {X 0,Y 233.135,Z 460.578,A -85,B 0,C 180,E1 -19697.818,E2 -19697.818} C_VEL
LIN {X 0,Y 232.707,Z 461.578,A -85,B 0,C 180,E1 -19701.315,E2 -19701.315} C_VEL
LIN {X 0,Y 232.694,Z 461.502,A -85,B 0,C 180,E1 -19703.061,E2 -19703.061} C_VEL
LIN {X 0,Y 232.715,Z 460.795,A -85,B 0,C 180,E1 -19705.281,E2 -19705.281} C_VEL
LIN {X 0,Y 232.869,Z 458.83,A -85,B 0,C 180,E1 -19708.27,E2 -19708.27} C_VEL
LIN {X 0,Y 233.166,Z 456.113,A -85,B 0,C 180,E1 -19710.863,E2 -19710.863} C_VEL
LIN {X 0,Y 233.699,Z 452.392,A -85,B 0,C 180,E1 -19713.448,E2 -19713.448} C_VEL
LIN {X 0,Y 234.625,Z 447.557,A -85,B 0,C 180,E1 -19716.018,E2 -19716.018} C_VEL
LIN {X 0,Y 235.816,Z 441.472,A -85,B 0,C 180,E1 -19718.57,E2 -19718.57} C_VEL
LIN {X 0,Y 237.47,Z 433.904,A -85,B 0,C 180,E1 -19721.091,E2 -19721.091} C_VEL
LIN {X 0,Y 239.444,Z 424.393,A -85,B 0,C 180,E1 -19723.58,E2 -19723.58} C_VEL
LIN {X 0,Y 241.415,Z 414.581,A -85,B 0,C 180,E1 -19725.622,E2 -19725.622} C_VEL
LIN {X 0,Y 243.374,Z 403.65,A -85,B 0,C 180,E1 -19727.421,E2 -19727.421} C_VEL
LIN {X 0,Y 245.142,Z 391.721,A -85,B 0,C 180,E1 -19728.948,E2 -19728.948} C_VEL
LIN {X 0,Y 246.608,Z 379.792,A -85,B 0,C 180,E1 -19730.106,E2 -19730.106} C_VEL
LIN {X 0,Y 247.702,Z 367.119,A -85,B 0,C 180,E1 -19730.99,E2 -19730.99} C_VEL
LIN {X 0,Y 248.48,Z 353.741,A -85,B 0,C 180,E1 -19731.573,E2 -19731.573} C_VEL
LIN {X 0,Y 250.735,Z 288.342,A -85,B 0,C 180,E1 -19733.386,E2 -19733.386} C_VEL
LIN {X 0,Y 244.746,Z 272.181,A -85,B 0,C 180,E1 -19734.627,E2 -19734.627} C_VEL
LIN {X 0,Y 236.762,Z 254.246,A -85,B 0,C 180,E1 -19736.28,E2 -19736.28} C_VEL
LIN {X 0,Y 235.162,Z 251.18,A -85,B 0,C 180,E1 -19736.609,E2 -19736.609} C_VEL
LIN {X 0,Y 235.025,Z 250.631,A -85,B 0,C 180,E1 -19736.65,E2 -19736.65} C_VEL
LIN {X 0,Y 234.959,Z 250.219,A -85,B 0,C 180,E1 -19736.899,E2 -19736.899} C_VEL
LIN {X 0,Y 234.901,Z 250.226,A -85,B 0,C 180,E1 -19740.572,E2 -19740.572} C_VEL
LIN {X 0,Y 234.932,Z 250.221,A -85,B 0,C 180,E1 -19744.638,E2 -19744.638} C_VEL
LIN {X 0,Y 234.943,Z 250.219,A -85,B 0,C 180,E1 -19748.944,E2 -19748.944} C_VEL
LIN {X 0,Y 234.891,Z 250.224,A -85,B 0,C 180,E1 -19753.485,E2 -19753.485} C_VEL
LIN {X 0,Y 234.891,Z 250.226,A -85,B 0,C 180,E1 -19756.514,E2 -19756.514} C_VEL
LIN {X 0,Y 234.919,Z 250.219,A -85,B 0,C 180,E1 -19761.078,E2 -19761.078} C_VEL
LIN {X 0,Y 234.932,Z 250.214,A -85,B 0,C 180,E1 -19765.362,E2 -19765.362} C_VEL
LIN {X 0,Y 234.923,Z 250.213,A -85,B 0,C 180,E1 -19769.431,E2 -19769.431} C_VEL
LIN {X 0,Y 234.995,Z 250.21,A -85,B 0,C 180,E1 -19773.794,E2 -19773.794} C_VEL
LIN {X 0,Y 235.013,Z 250.19,A -85,B 0,C 180,E1 -19778.97,E2 -19778.97} C_VEL
LIN {X 0,Y 235.098,Z 250.197,A -85,B 0,C 180,E1 -19783.059,E2 -19783.059} C_VEL
LIN {X 0,Y 235.115,Z 250.172,A -85,B 0,C 180,E1 -19787.922,E2 -19787.922} C_VEL
LIN {X 0,Y 235.313,Z 250.161,A -85,B 0,C 180,E1 -19791.412,E2 -19791.412} C_VEL
LIN {X 0,Y 235.206,Z 250.185,A -85,B 0,C 180,E1 -19794.857,E2 -19794.857} C_VEL
LIN {X 0,Y 235.595,Z 250.13,A -85,B 0,C 180,E1 -19798.29,E2 -19798.29} C_VEL
LIN {X 0,Y 235.595,Z 250.135,A -85,B 0,C 180,E1 -19801.709,E2 -19801.709} C_VEL
LIN {X 0,Y 235.406,Z 250.163,A -85,B 0,C 180,E1 -19806.858,E2 -19806.858} C_VEL
LIN {X 0,Y 235.254,Z 250.171,A -85,B 0,C 180,E1 -19810.326,E2 -19810.326} C_VEL
LIN {X 0,Y 235.075,Z 250.201,A -85,B 0,C 180,E1 -19815.609,E2 -19815.609} C_VEL
LIN {X 0,Y 234.971,Z 250.205,A -85,B 0,C 180,E1 -19818.287,E2 -19818.287} C_VEL
LIN {X 0,Y 234.288,Z 250.294,A -85,B 0,C 180,E1 -19819.717,E2 -19819.717} C_VEL
LIN {X 0,Y 231.422,Z 250.657,A -85,B 0,C 180,E1 -19822.051,E2 -19822.051} C_VEL
LIN {X 0,Y 229.002,Z 250.956,A -85,B 0,C 180,E1 -19823.954,E2 -19823.954} C_VEL
LIN {X 0,Y 227.978,Z 251.08,A -85,B 0,C 180,E1 -19825.431,E2 -19825.431} C_VEL
LIN {X 0,Y 227.901,Z 251.09,A -85,B 0,C 180,E1 -19825.932,E2 -19825.932} C_VEL
LIN {X 0,Y 227.874,Z 251.094,A -85,B 0,C 180,E1 -19830.281,E2 -19830.281} C_VEL
LIN {X 0,Y 227.877,Z 251.098,A -85,B 0,C 180,E1 -19833.72,E2 -19833.72} C_VEL
LIN {X 0,Y 227.843,Z 251.103,A -85,B 0,C 180,E1 -19838.091,E2 -19838.091} C_VEL
LIN {X 0,Y 227.801,Z 251.108,A -85,B 0,C 180,E1 -19842.745,E2 -19842.745} C_VEL
LIN {X 0,Y 227.81,Z 251.103,A -85,B 0,C 180,E1 -19847.257,E2 -19847.257} C_VEL
LIN {X 0,Y 227.948,Z 251.157,A -85,B 0,C 180,E1 -19852.108,E2 -19852.108} C_VEL
LIN {X 0,Y 229.811,Z 259.073,A -85,B 0,C 180,E1 -19855.66,E2 -19855.66} C_VEL
LIN {X 0,Y 230.312,Z 261.449,A -85,B 0,C 180,E1 -19856.683,E2 -19856.683} C_VEL
LIN {X 0,Y 238.618,Z 281.491,A -85,B 0,C 180,E1 -19858.542,E2 -19858.542} C_VEL
LIN {X 0,Y 240.257,Z 286.288,A -85,B 0,C 180,E1 -19858.915,E2 -19858.915} C_VEL
LIN {X 0,Y 243.634,Z 312.541,A -85,B 0,C 180,E1 -19860.197,E2 -19860.197} C_VEL
LIN {X 0,Y 241.565,Z 370.802,A -85,B 0,C 180,E1 -19861.899,E2 -19861.899} C_VEL
LIN {X 0,Y 240.453,Z 383.921,A -85,B 0,C 180,E1 -19862.591,E2 -19862.591} C_VEL
LIN {X 0,Y 238.972,Z 396.528,A -85,B 0,C 180,E1 -19863.588,E2 -19863.588} C_VEL
LIN {X 0,Y 237.294,Z 407.729,A -85,B 0,C 180,E1 -19864.802,E2 -19864.802} C_VEL
LIN {X 0,Y 235.264,Z 419.373,A -85,B 0,C 180,E1 -19866.45,E2 -19866.45} C_VEL
LIN {X 0,Y 233.055,Z 429.834,A -85,B 0,C 180,E1 -19868.321,E2 -19868.321} C_VEL
LIN {X 0,Y 231.222,Z 439.255,A -85,B 0,C 180,E1 -19870.467,E2 -19870.467} C_VEL
LIN {X 0,Y 230.017,Z 445.555,A -85,B 0,C 180,E1 -19872.209,E2 -19872.209} C_VEL
LIN {X 0,Y 228.312,Z 453.42,A -85,B 0,C 180,E1 -19874.832,E2 -19874.832} C_VEL
LIN {X 0,Y 227.035,Z 459.702,A -85,B 0,C 180,E1 -19877.485,E2 -19877.485} C_VEL
LIN {X 0,Y 226.279,Z 464.699,A -85,B 0,C 180,E1 -19880.164,E2 -19880.164} C_VEL
LIN {X 0,Y 225.821,Z 468.551,A -85,B 0,C 180,E1 -19882.849,E2 -19882.849} C_VEL
LIN {X 0,Y 225.625,Z 471.251,A -85,B 0,C 180,E1 -19885.393,E2 -19885.393} C_VEL
LIN {X 0,Y 225.666,Z 473.22,A -85,B 0,C 180,E1 -19888.215,E2 -19888.215} C_VEL
LIN {X 0,Y 225.734,Z 473.921,A -85,B 0,C 180,E1 -19890,E2 -19890} C_VEL
LIN {X 0,Y 225.656,Z 474.228,A -85,B 0,C 180,E1 -19891.785,E2 -19891.785} C_VEL
LIN {X 0,Y 225.597,Z 473.923,A -85,B 0,C 180,E1 -19894.518,E2 -19894.518} C_VEL
LIN {X 0,Y 225.826,Z 472.759,A -85,B 0,C 180,E1 -19897.151,E2 -19897.151} C_VEL
LIN {X 0,Y 226.664,Z 469.771,A -85,B 0,C 180,E1 -19900.722,E2 -19900.722} C_VEL
LIN {X 0,Y 227.725,Z 466.378,A -85,B 0,C 180,E1 -19903.383,E2 -19903.383} C_VEL
LIN {X 0,Y 229.294,Z 461.927,A -85,B 0,C 180,E1 -19906.013,E2 -19906.013} C_VEL
LIN {X 0,Y 231.387,Z 456.293,A -85,B 0,C 180,E1 -19908.598,E2 -19908.598} C_VEL
LIN {X 0,Y 233.804,Z 449.258,A -85,B 0,C 180,E1 -19911.144,E2 -19911.144} C_VEL
LIN {X 0,Y 236.571,Z 440.487,A -85,B 0,C 180,E1 -19913.644,E2 -19913.644} C_VEL
LIN {X 0,Y 239.739,Z 430.54,A -85,B 0,C 180,E1 -19915.853,E2 -19915.853} C_VEL
LIN {X 0,Y 242.551,Z 420.408,A -85,B 0,C 180,E1 -19917.62,E2 -19917.62} C_VEL
LIN {X 0,Y 245.298,Z 409.178,A -85,B 0,C 180,E1 -19919.148,E2 -19919.148} C_VEL
LIN {X 0,Y 247.848,Z 396.551,A -85,B 0,C 180,E1 -19920.455,E2 -19920.455} C_VEL
LIN {X 0,Y 249.81,Z 383.457,A -85,B 0,C 180,E1 -19921.423,E2 -19921.423} C_VEL
LIN {X 0,Y 251.207,Z 370.489,A -85,B 0,C 180,E1 -19922.052,E2 -19922.052} C_VEL
LIN {X 0,Y 253.367,Z 324.949,A -85,B 0,C 180,E1 -19923.321,E2 -19923.321} C_VEL
LIN {X 0,Y 253.503,Z 316.412,A -85,B 0,C 180,E1 -19923.591,E2 -19923.591} C_VEL
LIN {X 0,Y 251.264,Z 302.46,A -85,B 0,C 180,E1 -19924.451,E2 -19924.451} C_VEL
LIN {X 0,Y 245.464,Z 289.111,A -85,B 0,C 180,E1 -19925.962,E2 -19925.962} C_VEL
LIN {X 0,Y 238.349,Z 274.637,A -85,B 0,C 180,E1 -19927.892,E2 -19927.892} C_VEL
LIN {X 0,Y 232.898,Z 265.021,A -85,B 0,C 180,E1 -19929.432,E2 -19929.432} C_VEL
LIN {X 0,Y 230.52,Z 260.602,A -85,B 0,C 180,E1 -19930.213,E2 -19930.213} C_VEL
LIN {X 0,Y 228.641,Z 254.076,A -85,B 0,C 180,E1 -19933.751,E2 -19933.751} C_VEL
LIN {X 0,Y 227.84,Z 251.105,A -85,B 0,C 180,E1 -19935.51,E2 -19935.51} C_VEL
LIN {X 0,Y 227.829,Z 251.104,A -85,B 0,C 180,E1 -19940.461,E2 -19940.461} C_VEL
LIN {X 0,Y 227.866,Z 251.097,A -85,B 0,C 180,E1 -19944.125,E2 -19944.125} C_VEL
LIN {X 0,Y 227.857,Z 251.101,A -85,B 0,C 180,E1 -19948.376,E2 -19948.376} C_VEL
LIN {X 0,Y 227.858,Z 251.102,A -85,B 0,C 180,E1 -19952.441,E2 -19952.441} C_VEL
LIN {X 0,Y 227.899,Z 251.097,A -85,B 0,C 180,E1 -19956.366,E2 -19956.366} C_VEL
LIN {X 0,Y 227.925,Z 251.091,A -85,B 0,C 180,E1 -19960.173,E2 -19960.173} C_VEL
LIN {X 0,Y 228.025,Z 251.071,A -85,B 0,C 180,E1 -19963.896,E2 -19963.896} C_VEL
LIN {X 0,Y 228.071,Z 251.064,A -85,B 0,C 180,E1 -19967.543,E2 -19967.543} C_VEL
LIN {X 0,Y 228.307,Z 251.044,A -85,B 0,C 180,E1 -19971.146,E2 -19971.146} C_VEL
LIN {X 0,Y 228.354,Z 251.026,A -85,B 0,C 180,E1 -19972.929,E2 -19972.929} C_VEL
LIN {X 0,Y 228.55,Z 251.001,A -85,B 0,C 180,E1 -19978.238,E2 -19978.238} C_VEL
LIN {X 0,Y 228.552,Z 251.009,A -85,B 0,C 180,E1 -19981.762,E2 -19981.762} C_VEL
LIN {X 0,Y 228.305,Z 251.039,A -85,B 0,C 180,E1 -19987.073,E2 -19987.073} C_VEL
LIN {X 0,Y 228.143,Z 251.066,A -85,B 0,C 180,E1 -19990.652,E2 -19990.652} C_VEL
LIN {X 0,Y 228.044,Z 251.076,A -85,B 0,C 180,E1 -19996.103,E2 -19996.103} C_VEL
LIN {X 0,Y 227.939,Z 251.089,A -85,B 0,C 180,E1 -19999.826,E2 -19999.826} C_VEL
LIN {X 0,Y 227.916,Z 251.087,A -85,B 0,C 180,E1 -20003.633,E2 -20003.633} C_VEL
LIN {X 0,Y 227.888,Z 251.092,A -85,B 0,C 180,E1 -20007.555,E2 -20007.555} C_VEL
LIN {X 0,Y 227.875,Z 251.1,A -85,B 0,C 180,E1 -20011.622,E2 -20011.622} C_VEL
LIN {X 0,Y 227.902,Z 251.092,A -85,B 0,C 180,E1 -20015.868,E2 -20015.868} C_VEL
LIN {X 0,Y 227.835,Z 251.106,A -85,B 0,C 180,E1 -20020.375,E2 -20020.375} C_VEL
LIN {X 0,Y 227.83,Z 251.121,A -85,B 0,C 180,E1 -20023.04,E2 -20023.04} C_VEL
LIN {X 0,Y 227.967,Z 251.836,A -85,B 0,C 180,E1 -20023.311,E2 -20023.311} C_VEL
LIN {X 0,Y 229.306,Z 254.582,A -85,B 0,C 180,E1 -20023.745,E2 -20023.745} C_VEL
LIN {X 0,Y 230.942,Z 256.461,A -85,B 0,C 180,E1 -20024.203,E2 -20024.203} C_VEL
LIN {X 0,Y 237.031,Z 266.419,A -85,B 0,C 180,E1 -20025.941,E2 -20025.941} C_VEL
LIN {X 0,Y 244.35,Z 279.605,A -85,B 0,C 180,E1 -20027.905,E2 -20027.905} C_VEL
LIN {X 0,Y 251.523,Z 294.631,A -85,B 0,C 180,E1 -20029.745,E2 -20029.745} C_VEL
LIN {X 0,Y 254.332,Z 301.352,A -85,B 0,C 180,E1 -20030.454,E2 -20030.454} C_VEL
LIN {X 0,Y 251.662,Z 358.992,A -85,B 0,C 180,E1 -20032.055,E2 -20032.055} C_VEL
LIN {X 0,Y 250.394,Z 372.588,A -85,B 0,C 180,E1 -20032.756,E2 -20032.756} C_VEL
LIN {X 0,Y 248.583,Z 385.094,A -85,B 0,C 180,E1 -20033.704,E2 -20033.704} C_VEL
LIN {X 0,Y 246.331,Z 397.031,A -85,B 0,C 180,E1 -20034.958,E2 -20034.958} C_VEL
LIN {X 0,Y 243.682,Z 408.473,A -85,B 0,C 180,E1 -20036.524,E2 -20036.524} C_VEL
LIN {X 0,Y 241.35,Z 417.373,A -85,B 0,C 180,E1 -20038.069,E2 -20038.069} C_VEL
LIN {X 0,Y 238.569,Z 426.275,A -85,B 0,C 180,E1 -20039.947,E2 -20039.947} C_VEL
LIN {X 0,Y 236.071,Z 434.163,A -85,B 0,C 180,E1 -20042.038,E2 -20042.038} C_VEL
LIN {X 0,Y 233.447,Z 441.788,A -85,B 0,C 180,E1 -20044.578,E2 -20044.578} C_VEL
LIN {X 0,Y 230.826,Z 448.877,A -85,B 0,C 180,E1 -20047.63,E2 -20047.63} C_VEL
LIN {X 0,Y 229.051,Z 453.532,A -85,B 0,C 180,E1 -20050.274,E2 -20050.274} C_VEL
LIN {X 0,Y 227.59,Z 457.342,A -85,B 0,C 180,E1 -20053.194,E2 -20053.194} C_VEL
LIN {X 0,Y 226.661,Z 459.567,A -85,B 0,C 180,E1 -20055.638,E2 -20055.638} C_VEL
LIN {X 0,Y 226.133,Z 460.726,A -85,B 0,C 180,E1 -20057.435,E2 -20057.435} C_VEL
LIN {X 0,Y 225.637,Z 461.767,A -85,B 0,C 180,E1 -20061.04,E2 -20061.04} C_VEL
LIN {X 0,Y 225.591,Z 461.71,A -85,B 0,C 180,E1 -20062.841,E2 -20062.841} C_VEL
LIN {X 0,Y 225.621,Z 460.913,A -85,B 0,C 180,E1 -20065.412,E2 -20065.412} C_VEL
LIN {X 0,Y 225.775,Z 459.112,A -85,B 0,C 180,E1 -20068.216,E2 -20068.216} C_VEL
LIN {X 0,Y 226.087,Z 456.434,A -85,B 0,C 180,E1 -20070.891,E2 -20070.891} C_VEL
LIN {X 0,Y 226.63,Z 452.756,A -85,B 0,C 180,E1 -20073.556,E2 -20073.556} C_VEL
LIN {X 0,Y 227.58,Z 447.966,A -85,B 0,C 180,E1 -20076.205,E2 -20076.205} C_VEL
LIN {X 0,Y 228.818,Z 441.931,A -85,B 0,C 180,E1 -20078.834,E2 -20078.834} C_VEL
LIN {X 0,Y 230.533,Z 434.424,A -85,B 0,C 180,E1 -20081.429,E2 -20081.429} C_VEL
LIN {X 0,Y 232.323,Z 426.748,A -85,B 0,C 180,E1 -20083.559,E2 -20083.559} C_VEL
LIN {X 0,Y 234.411,Z 416.341,A -85,B 0,C 180,E1 -20085.877,E2 -20085.877} C_VEL
LIN {X 0,Y 236.311,Z 406.42,A -85,B 0,C 180,E1 -20087.63,E2 -20087.63} C_VEL
LIN {X 0,Y 238.028,Z 395.802,A -85,B 0,C 180,E1 -20089.134,E2 -20089.134} C_VEL
LIN {X 0,Y 239.592,Z 384.621,A -85,B 0,C 180,E1 -20090.363,E2 -20090.363} C_VEL
LIN {X 0,Y 240.882,Z 371.974,A -85,B 0,C 180,E1 -20091.389,E2 -20091.389} C_VEL
LIN {X 0,Y 241.779,Z 359.198,A -85,B 0,C 180,E1 -20092.09,E2 -20092.09} C_VEL
LIN {X 0,Y 243.352,Z 320.145,A -85,B 0,C 180,E1 -20093.237,E2 -20093.237} C_VEL
LIN {X 0,Y 244.312,Z 289.615,A -85,B 0,C 180,E1 -20094.113,E2 -20094.113} C_VEL
LIN {X 0,Y 238.288,Z 273.695,A -85,B 0,C 180,E1 -20095.411,E2 -20095.411} C_VEL
LIN {X 0,Y 231.417,Z 258.173,A -85,B 0,C 180,E1 -20096.902,E2 -20096.902} C_VEL
LIN {X 0,Y 228.224,Z 252.486,A -85,B 0,C 180,E1 -20097.578,E2 -20097.578} C_VEL
LIN {X 0,Y 227.909,Z 251.096,A -85,B 0,C 180,E1 -20097.708,E2 -20097.708} C_VEL
LIN {X 0,Y 227.858,Z 251.102,A -85,B 0,C 180,E1 -20101.624,E2 -20101.624} C_VEL
LIN {X 0,Y 227.883,Z 251.097,A -85,B 0,C 180,E1 -20105.871,E2 -20105.871} C_VEL
LIN {X 0,Y 227.828,Z 251.105,A -85,B 0,C 180,E1 -20110.376,E2 -20110.376} C_VEL
LIN {X 0,Y 227.837,Z 251.104,A -85,B 0,C 180,E1 -20115.192,E2 -20115.192} C_VEL
LIN {X 0,Y 227.828,Z 251.104,A -85,B 0,C 180,E1 -20119.623,E2 -20119.623} C_VEL
LIN {X 0,Y 227.882,Z 251.099,A -85,B 0,C 180,E1 -20124.128,E2 -20124.128} C_VEL
LIN {X 0,Y 227.868,Z 251.08,A -85,B 0,C 180,E1 -20128.377,E2 -20128.377} C_VEL
LIN {X 0,Y 227.88,Z 251.099,A -85,B 0,C 180,E1 -20132.444,E2 -20132.444} C_VEL
LIN {X 0,Y 227.915,Z 251.073,A -85,B 0,C 180,E1 -20136.367,E2 -20136.367} C_VEL
LIN {X 0,Y 227.944,Z 251.078,A -85,B 0,C 180,E1 -20140.174,E2 -20140.174} C_VEL
LIN {X 0,Y 228.059,Z 251.073,A -85,B 0,C 180,E1 -20143.898,E2 -20143.898} C_VEL
LIN {X 0,Y 228.073,Z 251.051,A -85,B 0,C 180,E1 -20147.543,E2 -20147.543} C_VEL
LIN {X 0,Y 228.254,Z 251.035,A -85,B 0,C 180,E1 -20151.144,E2 -20151.144} C_VEL
LIN {X 0,Y 228.304,Z 251.041,A -85,B 0,C 180,E1 -20152.927,E2 -20152.927} C_VEL
LIN {X 0,Y 228.553,Z 251.006,A -85,B 0,C 180,E1 -20158.238,E2 -20158.238} C_VEL
LIN {X 0,Y 228.553,Z 251.013,A -85,B 0,C 180,E1 -20161.762,E2 -20161.762} C_VEL
LIN {X 0,Y 228.359,Z 251.039,A -85,B 0,C 180,E1 -20167.071,E2 -20167.071} C_VEL
LIN {X 0,Y 228.167,Z 251.051,A -85,B 0,C 180,E1 -20170.65,E2 -20170.65} C_VEL
LIN {X 0,Y 228.042,Z 251.077,A -85,B 0,C 180,E1 -20174.273,E2 -20174.273} C_VEL
LIN {X 0,Y 227.93,Z 251.082,A -85,B 0,C 180,E1 -20178.26,E2 -20178.26} C_VEL
LIN {X 0,Y 227.92,Z 251.095,A -85,B 0,C 180,E1 -20182.323,E2 -20182.323} C_VEL
LIN {X 0,Y 227.901,Z 251.09,A -85,B 0,C 180,E1 -20185.932,E2 -20185.932} C_VEL
LIN {X 0,Y 227.238,Z 251.179,A -85,B 0,C 180,E1 -20187.407,E2 -20187.407} C_VEL
LIN {X 0,Y 224.35,Z 251.538,A -85,B 0,C 180,E1 -20189.812,E2 -20189.812} C_VEL
LIN {X 0,Y 221.901,Z 251.842,A -85,B 0,C 180,E1 -20191.775,E2 -20191.775} C_VEL
LIN {X 0,Y 220.869,Z 251.971,A -85,B 0,C 180,E1 -20193.301,E2 -20193.301} C_VEL
LIN {X 0,Y 220.797,Z 251.979,A -85,B 0,C 180,E1 -20193.818,E2 -20193.818} C_VEL
LIN {X 0,Y 220.81,Z 251.979,A -85,B 0,C 180,E1 -20197.278,E2 -20197.278} C_VEL
LIN {X 0,Y 220.759,Z 251.984,A -85,B 0,C 180,E1 -20201.955,E2 -20201.955} C_VEL
LIN {X 0,Y 220.77,Z 251.982,A -85,B 0,C 180,E1 -20205.545,E2 -20205.545} C_VEL
LIN {X 0,Y 220.808,Z 251.98,A -85,B 0,C 180,E1 -20210.463,E2 -20210.463} C_VEL
LIN {X 0,Y 220.862,Z 252.107,A -85,B 0,C 180,E1 -20211.323,E2 -20211.323} C_VEL
LIN {X 0,Y 223.064,Z 261.226,A -85,B 0,C 180,E1 -20215.576,E2 -20215.576} C_VEL
LIN {X 0,Y 231.032,Z 279.882,A -85,B 0,C 180,E1 -20217.454,E2 -20217.454} C_VEL
LIN {X 0,Y 234.18,Z 288.397,A -85,B 0,C 180,E1 -20218.185,E2 -20218.185} C_VEL
LIN {X 0,Y 237.314,Z 313.323,A -85,B 0,C 180,E1 -20219.443,E2 -20219.443} C_VEL
LIN {X 0,Y 235.201,Z 370.327,A -85,B 0,C 180,E1 -20221.143,E2 -20221.143} C_VEL
LIN {X 0,Y 234.078,Z 383.367,A -85,B 0,C 180,E1 -20221.84,E2 -20221.84} C_VEL
LIN {X 0,Y 232.63,Z 395.508,A -85,B 0,C 180,E1 -20222.81,E2 -20222.81} C_VEL
LIN {X 0,Y 230.856,Z 406.941,A -85,B 0,C 180,E1 -20224.048,E2 -20224.048} C_VEL
LIN {X 0,Y 228.722,Z 418.697,A -85,B 0,C 180,E1 -20225.734,E2 -20225.734} C_VEL
LIN {X 0,Y 226.468,Z 429.244,A -85,B 0,C 180,E1 -20227.657,E2 -20227.657} C_VEL
LIN {X 0,Y 224.378,Z 439.269,A -85,B 0,C 180,E1 -20229.995,E2 -20229.995} C_VEL
LIN {X 0,Y 222.877,Z 446.54,A -85,B 0,C 180,E1 -20232.095,E2 -20232.095} C_VEL
LIN {X 0,Y 221.191,Z 454.143,A -85,B 0,C 180,E1 -20234.804,E2 -20234.804} C_VEL
LIN {X 0,Y 219.76,Z 461.166,A -85,B 0,C 180,E1 -20238.002,E2 -20238.002} C_VEL
LIN {X 0,Y 219.053,Z 465.807,A -85,B 0,C 180,E1 -20240.769,E2 -20240.769} C_VEL
LIN {X 0,Y 218.759,Z 468.256,A -85,B 0,C 180,E1 -20242.617,E2 -20242.617} C_VEL
LIN {X 0,Y 218.548,Z 471.176,A -85,B 0,C 180,E1 -20245.481,E2 -20245.481} C_VEL
LIN {X 0,Y 218.563,Z 472.987,A -85,B 0,C 180,E1 -20248.157,E2 -20248.157} C_VEL
LIN {X 0,Y 218.648,Z 473.703,A -85,B 0,C 180,E1 -20250,E2 -20250} C_VEL
LIN {X 0,Y 218.553,Z 474.024,A -85,B 0,C 180,E1 -20251.843,E2 -20251.843} C_VEL
LIN {X 0,Y 218.513,Z 473.819,A -85,B 0,C 180,E1 -20254.403,E2 -20254.403} C_VEL
LIN {X 0,Y 218.765,Z 472.614,A -85,B 0,C 180,E1 -20257.383,E2 -20257.383} C_VEL
LIN {X 0,Y 219.671,Z 469.656,A -85,B 0,C 180,E1 -20261.067,E2 -20261.067} C_VEL
LIN {X 0,Y 220.774,Z 466.295,A -85,B 0,C 180,E1 -20263.813,E2 -20263.813} C_VEL
LIN {X 0,Y 222.457,Z 461.878,A -85,B 0,C 180,E1 -20266.519,E2 -20266.519} C_VEL
LIN {X 0,Y 224.623,Z 456.281,A -85,B 0,C 180,E1 -20269.179,E2 -20269.179} C_VEL
LIN {X 0,Y 227.347,Z 448.763,A -85,B 0,C 180,E1 -20271.968,E2 -20271.968} C_VEL
LIN {X 0,Y 230.088,Z 440.589,A -85,B 0,C 180,E1 -20274.353,E2 -20274.353} C_VEL
LIN {X 0,Y 233.071,Z 431.676,A -85,B 0,C 180,E1 -20276.409,E2 -20276.409} C_VEL
LIN {X 0,Y 235.969,Z 421.894,A -85,B 0,C 180,E1 -20278.217,E2 -20278.217} C_VEL
LIN {X 0,Y 238.792,Z 411.139,A -85,B 0,C 180,E1 -20279.779,E2 -20279.779} C_VEL
LIN {X 0,Y 241.384,Z 399.082,A -85,B 0,C 180,E1 -20281.118,E2 -20281.118} C_VEL
LIN {X 0,Y 243.537,Z 386.5,A -85,B 0,C 180,E1 -20282.145,E2 -20282.145} C_VEL
LIN {X 0,Y 245.028,Z 374.243,A -85,B 0,C 180,E1 -20282.839,E2 -20282.839} C_VEL
LIN {X 0,Y 246.074,Z 359.735,A -85,B 0,C 180,E1 -20283.317,E2 -20283.317} C_VEL
LIN {X 0,Y 247.833,Z 318.007,A -85,B 0,C 180,E1 -20284.494,E2 -20284.494} C_VEL
LIN {X 0,Y 245.806,Z 305.171,A -85,B 0,C 180,E1 -20285.314,E2 -20285.314} C_VEL
LIN {X 0,Y 239.517,Z 290.685,A -85,B 0,C 180,E1 -20287.04,E2 -20287.04} C_VEL
LIN {X 0,Y 233.12,Z 277.869,A -85,B 0,C 180,E1 -20288.864,E2 -20288.864} C_VEL
LIN {X 0,Y 228.441,Z 269.538,A -85,B 0,C 180,E1 -20290.255,E2 -20290.255} C_VEL
LIN {X 0,Y 225.471,Z 264.51,A -85,B 0,C 180,E1 -20291.174,E2 -20291.174} C_VEL
LIN {X 0,Y 223.23,Z 260.451,A -85,B 0,C 180,E1 -20291.916,E2 -20291.916} C_VEL
LIN {X 0,Y 220.785,Z 251.984,A -85,B 0,C 180,E1 -20296.939,E2 -20296.939} C_VEL
LIN {X 0,Y 220.784,Z 251.982,A -85,B 0,C 180,E1 -20300.458,E2 -20300.458} C_VEL
LIN {X 0,Y 220.825,Z 251.969,A -85,B 0,C 180,E1 -20302.793,E2 -20302.793} C_VEL
LIN {X 0,Y 220.813,Z 251.97,A -85,B 0,C 180,E1 -20307.243,E2 -20307.243} C_VEL
LIN {X 0,Y 220.806,Z 251.973,A -85,B 0,C 180,E1 -20311.482,E2 -20311.482} C_VEL
LIN {X 0,Y 220.85,Z 251.968,A -85,B 0,C 180,E1 -20315.563,E2 -20315.563} C_VEL
LIN {X 0,Y 220.879,Z 251.962,A -85,B 0,C 180,E1 -20319.513,E2 -20319.513} C_VEL
LIN {X 0,Y 220.98,Z 251.948,A -85,B 0,C 180,E1 -20323.368,E2 -20323.368} C_VEL
LIN {X 0,Y 221.107,Z 251.933,A -85,B 0,C 180,E1 -20329.006,E2 -20329.006} C_VEL
LIN {X 0,Y 221.29,Z 251.906,A -85,B 0,C 180,E1 -20332.702,E2 -20332.702} C_VEL
LIN {X 0,Y 221.508,Z 251.878,A -85,B 0,C 180,E1 -20338.182,E2 -20338.182} C_VEL
LIN {X 0,Y 221.51,Z 251.886,A -85,B 0,C 180,E1 -20341.818,E2 -20341.818} C_VEL
LIN {X 0,Y 221.242,Z 251.916,A -85,B 0,C 180,E1 -20347.3,E2 -20347.3} C_VEL
LIN {X 0,Y 221.064,Z 251.949,A -85,B 0,C 180,E1 -20350.997,E2 -20350.997} C_VEL
LIN {X 0,Y 221.008,Z 251.951,A -85,B 0,C 180,E1 -20356.631,E2 -20356.631} C_VEL
LIN {X 0,Y 220.891,Z 251.967,A -85,B 0,C 180,E1 -20360.487,E2 -20360.487} C_VEL
LIN {X 0,Y 220.869,Z 251.971,A -85,B 0,C 180,E1 -20364.435,E2 -20364.435} C_VEL
LIN {X 0,Y 220.839,Z 251.976,A -85,B 0,C 180,E1 -20368.514,E2 -20368.514} C_VEL
LIN {X 0,Y 220.826,Z 251.974,A -85,B 0,C 180,E1 -20372.755,E2 -20372.755} C_VEL
LIN {X 0,Y 220.84,Z 251.974,A -85,B 0,C 180,E1 -20377.288,E2 -20377.288} C_VEL
LIN {X 0,Y 220.775,Z 251.981,A -85,B 0,C 180,E1 -20381.469,E2 -20381.469} C_VEL
LIN {X 0,Y 221.728,Z 254.777,A -85,B 0,C 180,E1 -20381.886,E2 -20381.886} C_VEL
LIN {X 0,Y 223.994,Z 257.414,A -85,B 0,C 180,E1 -20382.58,E2 -20382.58} C_VEL
LIN {X 0,Y 226.158,Z 260.723,A -85,B 0,C 180,E1 -20383.256,E2 -20383.256} C_VEL
LIN {X 0,Y 230.45,Z 267.359,A -85,B 0,C 180,E1 -20384.542,E2 -20384.542} C_VEL
LIN {X 0,Y 238.112,Z 280.838,A -85,B 0,C 180,E1 -20386.727,E2 -20386.727} C_VEL
LIN {X 0,Y 245.126,Z 295.368,A -85,B 0,C 180,E1 -20388.631,E2 -20388.631} C_VEL
LIN {X 0,Y 248.506,Z 303.251,A -85,B 0,C 180,E1 -20389.524,E2 -20389.524} C_VEL
LIN {X 0,Y 245.902,Z 358.885,A -85,B 0,C 180,E1 -20391.106,E2 -20391.106} C_VEL
LIN {X 0,Y 244.622,Z 372.115,A -85,B 0,C 180,E1 -20391.786,E2 -20391.786} C_VEL
LIN {X 0,Y 242.861,Z 384.263,A -85,B 0,C 180,E1 -20392.707,E2 -20392.707} C_VEL
LIN {X 0,Y 240.521,Z 396.483,A -85,B 0,C 180,E1 -20393.981,E2 -20393.981} C_VEL
LIN {X 0,Y 238.038,Z 406.754,A -85,B 0,C 180,E1 -20395.365,E2 -20395.365} C_VEL
LIN {X 0,Y 235.213,Z 417.273,A -85,B 0,C 180,E1 -20397.183,E2 -20397.183} C_VEL
LIN {X 0,Y 232.38,Z 426.049,A -85,B 0,C 180,E1 -20399.06,E2 -20399.06} C_VEL
LIN {X 0,Y 229.724,Z 434.011,A -85,B 0,C 180,E1 -20401.194,E2 -20401.194} C_VEL
LIN {X 0,Y 227.365,Z 440.593,A -85,B 0,C 180,E1 -20403.372,E2 -20403.372} C_VEL
LIN {X 0,Y 224.91,Z 447.041,A -85,B 0,C 180,E1 -20406.032,E2 -20406.032} C_VEL
LIN {X 0,Y 222.842,Z 452.134,A -85,B 0,C 180,E1 -20408.735,E2 -20408.735} C_VEL
LIN {X 0,Y 221.284,Z 456.069,A -85,B 0,C 180,E1 -20411.482,E2 -20411.482} C_VEL
LIN {X 0,Y 220.429,Z 458.084,A -85,B 0,C 180,E1 -20413.325,E2 -20413.325} C_VEL
LIN {X 0,Y 219.698,Z 459.679,A -85,B 0,C 180,E1 -20415.172,E2 -20415.172} C_VEL
LIN {X 0,Y 219.146,Z 460.868,A -85,B 0,C 180,E1 -20417.027,E2 -20417.027} C_VEL
LIN {X 0,Y 218.569,Z 461.955,A -85,B 0,C 180,E1 -20420.748,E2 -20420.748} C_VEL
LIN {X 0,Y 218.516,Z 461.917,A -85,B 0,C 180,E1 -20422.608,E2 -20422.608} C_VEL
LIN {X 0,Y 218.549,Z 461.061,A -85,B 0,C 180,E1 -20425.481,E2 -20425.481} C_VEL
LIN {X 0,Y 218.683,Z 459.393,A -85,B 0,C 180,E1 -20428.158,E2 -20428.158} C_VEL
LIN {X 0,Y 219.01,Z 456.755,A -85,B 0,C 180,E1 -20430.919,E2 -20430.919} C_VEL
LIN {X 0,Y 219.564,Z 453.119,A -85,B 0,C 180,E1 -20433.67,E2 -20433.67} C_VEL
LIN {X 0,Y 220.539,Z 448.375,A -85,B 0,C 180,E1 -20436.404,E2 -20436.404} C_VEL
LIN {X 0,Y 221.828,Z 442.389,A -85,B 0,C 180,E1 -20439.115,E2 -20439.115} C_VEL
LIN {X 0,Y 223.606,Z 434.938,A -85,B 0,C 180,E1 -20441.788,E2 -20441.788} C_VEL
LIN {X 0,Y 225.436,Z 427.329,A -85,B 0,C 180,E1 -20443.981,E2 -20443.981} C_VEL
LIN {X 0,Y 227.415,Z 418.102,A -85,B 0,C 180,E1 -20446.149,E2 -20446.149} C_VEL
LIN {X 0,Y 229.466,Z 407.957,A -85,B 0,C 180,E1 -20448.042,E2 -20448.042} C_VEL
LIN {X 0,Y 231.435,Z 396.439,A -85,B 0,C 180,E1 -20449.745,E2 -20449.745} C_VEL
LIN {X 0,Y 233.163,Z 384.541,A -85,B 0,C 180,E1 -20451.089,E2 -20451.089} C_VEL
LIN {X 0,Y 234.556,Z 371.325,A -85,B 0,C 180,E1 -20452.169,E2 -20452.169} C_VEL
LIN {X 0,Y 235.46,Z 358.566,A -85,B 0,C 180,E1 -20452.867,E2 -20452.867} C_VEL
LIN {X 0,Y 238.021,Z 291.359,A -85,B 0,C 180,E1 -20454.85,E2 -20454.85} C_VEL
LIN {X 0,Y 232.519,Z 276.71,A -85,B 0,C 180,E1 -20456.094,E2 -20456.094} C_VEL
LIN {X 0,Y 226.048,Z 262.107,A -85,B 0,C 180,E1 -20457.56,E2 -20457.56} C_VEL
LIN {X 0,Y 221.905,Z 254.932,A -85,B 0,C 180,E1 -20458.475,E2 -20458.475} C_VEL
LIN {X 0,Y 220.85,Z 251.976,A -85,B 0,C 180,E1 -20458.812,E2 -20458.812} C_VEL
LIN {X 0,Y 220.814,Z 251.98,A -85,B 0,C 180,E1 -20462.756,E2 -20462.756} C_VEL
LIN {X 0,Y 220.812,Z 251.979,A -85,B 0,C 180,E1 -20467.278,E2 -20467.278} C_VEL
LIN {X 0,Y 220.772,Z 251.982,A -85,B 0,C 180,E1 -20471.952,E2 -20471.952} C_VEL
LIN {X 0,Y 220.777,Z 251.982,A -85,B 0,C 180,E1 -20475.546,E2 -20475.546} C_VEL
LIN {X 0,Y 220.808,Z 251.979,A -85,B 0,C 180,E1 -20480.463,E2 -20480.463} C_VEL
LIN {X 0,Y 220.803,Z 251.975,A -85,B 0,C 180,E1 -20485.045,E2 -20485.045} C_VEL
LIN {X 0,Y 220.835,Z 251.964,A -85,B 0,C 180,E1 -20489.389,E2 -20489.389} C_VEL
LIN {X 0,Y 220.896,Z 251.966,A -85,B 0,C 180,E1 -20493.549,E2 -20493.549} C_VEL
LIN {X 0,Y 220.879,Z 251.941,A -85,B 0,C 180,E1 -20497.553,E2 -20497.553} C_VEL
LIN {X 0,Y 220.986,Z 251.956,A -85,B 0,C 180,E1 -20502.571,E2 -20502.571} C_VEL
LIN {X 0,Y 221.012,Z 251.931,A -85,B 0,C 180,E1 -20507.138,E2 -20507.138} C_VEL
LIN {X 0,Y 221.195,Z 251.91,A -85,B 0,C 180,E1 -20510.859,E2 -20510.859} C_VEL
LIN {X 0,Y 221.127,Z 251.938,A -85,B 0,C 180,E1 -20514.528,E2 -20514.528} C_VEL
LIN {X 0,Y 221.511,Z 251.882,A -85,B 0,C 180,E1 -20518.182,E2 -20518.182} C_VEL
LIN {X 0,Y 221.511,Z 251.89,A -85,B 0,C 180,E1 -20521.818,E2 -20521.818} C_VEL
LIN {X 0,Y 221.312,Z 251.916,A -85,B 0,C 180,E1 -20527.298,E2 -20527.298} C_VEL
LIN {X 0,Y 221.11,Z 251.928,A -85,B 0,C 180,E1 -20530.994,E2 -20530.994} C_VEL
LIN {X 0,Y 220.978,Z 251.954,A -85,B 0,C 180,E1 -20536.633,E2 -20536.633} C_VEL
LIN {X 0,Y 220.876,Z 251.967,A -85,B 0,C 180,E1 -20540.488,E2 -20540.488} C_VEL
LIN {X 0,Y 220.847,Z 251.968,A -85,B 0,C 180,E1 -20544.437,E2 -20544.437} C_VEL
LIN {X 0,Y 220.805,Z 251.981,A -85,B 0,C 180,E1 -20548.518,E2 -20548.518} C_VEL
LIN {X 0,Y 220.812,Z 251.981,A -85,B 0,C 180,E1 -20552.757,E2 -20552.757} C_VEL
LIN {X 0,Y 220.797,Z 251.979,A -85,B 0,C 180,E1 -20553.818,E2 -20553.818} C_VEL
LIN {X 0,Y 220.154,Z 252.06,A -85,B 0,C 180,E1 -20555.34,E2 -20555.34} C_VEL
LIN {X 0,Y 217.292,Z 252.419,A -85,B 0,C 180,E1 -20557.823,E2 -20557.823} C_VEL
LIN {X 0,Y 214.828,Z 252.724,A -85,B 0,C 180,E1 -20559.851,E2 -20559.851} C_VEL
LIN {X 0,Y 213.753,Z 252.857,A -85,B 0,C 180,E1 -20561.427,E2 -20561.427} C_VEL
LIN {X 0,Y 213.657,Z 252.864,A -85,B 0,C 180,E1 -20561.962,E2 -20561.962} C_VEL
LIN {X 0,Y 213.704,Z 252.865,A -85,B 0,C 180,E1 -20566.345,E2 -20566.345} C_VEL
LIN {X 0,Y 213.766,Z 252.86,A -85,B 0,C 180,E1 -20570.387,E2 -20570.387} C_VEL
LIN {X 0,Y 215.884,Z 261.277,A -85,B 0,C 180,E1 -20574.416,E2 -20574.416} C_VEL
LIN {X 0,Y 224.059,Z 279.751,A -85,B 0,C 180,E1 -20576.427,E2 -20576.427} C_VEL
LIN {X 0,Y 228.133,Z 290.674,A -85,B 0,C 180,E1 -20577.422,E2 -20577.422} C_VEL
LIN {X 0,Y 231.067,Z 314.777,A -85,B 0,C 180,E1 -20578.676,E2 -20578.676} C_VEL
LIN {X 0,Y 228.836,Z 370.398,A -85,B 0,C 180,E1 -20580.369,E2 -20580.369} C_VEL
LIN {X 0,Y 227.666,Z 383.574,A -85,B 0,C 180,E1 -20581.099,E2 -20581.099} C_VEL
LIN {X 0,Y 226.16,Z 395.611,A -85,B 0,C 180,E1 -20582.091,E2 -20582.091} C_VEL
LIN {X 0,Y 224.185,Z 407.759,A -85,B 0,C 180,E1 -20583.466,E2 -20583.466} C_VEL
LIN {X 0,Y 221.97,Z 419.323,A -85,B 0,C 180,E1 -20585.196,E2 -20585.196} C_VEL
LIN {X 0,Y 219.641,Z 429.728,A -85,B 0,C 180,E1 -20587.172,E2 -20587.172} C_VEL
LIN {X 0,Y 217.461,Z 439.641,A -85,B 0,C 180,E1 -20589.593,E2 -20589.593} C_VEL
LIN {X 0,Y 216.118,Z 446.092,A -85,B 0,C 180,E1 -20591.515,E2 -20591.515} C_VEL
LIN {X 0,Y 214.29,Z 453.739,A -85,B 0,C 180,E1 -20594.302,E2 -20594.302} C_VEL
LIN {X 0,Y 212.78,Z 460.802,A -85,B 0,C 180,E1 -20597.603,E2 -20597.603} C_VEL
LIN {X 0,Y 212.028,Z 465.481,A -85,B 0,C 180,E1 -20600.46,E2 -20600.46} C_VEL
LIN {X 0,Y 211.566,Z 469.034,A -85,B 0,C 180,E1 -20603.323,E2 -20603.323} C_VEL
LIN {X 0,Y 211.437,Z 471.57,A -85,B 0,C 180,E1 -20606.188,E2 -20606.188} C_VEL
LIN {X 0,Y 211.462,Z 472.75,A -85,B 0,C 180,E1 -20608.095,E2 -20608.095} C_VEL
LIN {X 0,Y 211.563,Z 473.484,A -85,B 0,C 180,E1 -20610,E2 -20610} C_VEL
LIN {X 0,Y 211.452,Z 473.819,A -85,B 0,C 180,E1 -20611.905,E2 -20611.905} C_VEL
LIN {X 0,Y 211.419,Z 473.72,A -85,B 0,C 180,E1 -20614.241,E2 -20614.241} C_VEL
LIN {X 0,Y 211.694,Z 472.468,A -85,B 0,C 180,E1 -20617.631,E2 -20617.631} C_VEL
LIN {X 0,Y 212.693,Z 469.541,A -85,B 0,C 180,E1 -20621.435,E2 -20621.435} C_VEL
LIN {X 0,Y 213.848,Z 466.211,A -85,B 0,C 180,E1 -20624.27,E2 -20624.27} C_VEL
LIN {X 0,Y 215.646,Z 461.829,A -85,B 0,C 180,E1 -20627.057,E2 -20627.057} C_VEL
LIN {X 0,Y 217.9,Z 456.27,A -85,B 0,C 180,E1 -20629.795,E2 -20629.795} C_VEL
LIN {X 0,Y 220.572,Z 449.349,A -85,B 0,C 180,E1 -20632.479,E2 -20632.479} C_VEL
LIN {X 0,Y 223.634,Z 440.695,A -85,B 0,C 180,E1 -20635.104,E2 -20635.104} C_VEL
LIN {X 0,Y 226.74,Z 431.844,A -85,B 0,C 180,E1 -20637.206,E2 -20637.206} C_VEL
LIN {X 0,Y 229.745,Z 422.136,A -85,B 0,C 180,E1 -20639.053,E2 -20639.053} C_VEL
LIN {X 0,Y 232.687,Z 411.51,A -85,B 0,C 180,E1 -20640.643,E2 -20640.643} C_VEL
LIN {X 0,Y 235.362,Z 399.627,A -85,B 0,C 180,E1 -20642.007,E2 -20642.007} C_VEL
LIN {X 0,Y 237.572,Z 387.275,A -85,B 0,C 180,E1 -20643.054,E2 -20643.054} C_VEL
LIN {X 0,Y 239.229,Z 374.56,A -85,B 0,C 180,E1 -20643.803,E2 -20643.803} C_VEL
LIN {X 0,Y 240.357,Z 359.907,A -85,B 0,C 180,E1 -20644.299,E2 -20644.299} C_VEL
LIN {X 0,Y 242.155,Z 319.223,A -85,B 0,C 180,E1 -20645.467,E2 -20645.467} C_VEL
LIN {X 0,Y 240.416,Z 307.992,A -85,B 0,C 180,E1 -20646.211,E2 -20646.211} C_VEL
LIN {X 0,Y 234.447,Z 294.129,A -85,B 0,C 180,E1 -20647.934,E2 -20647.934} C_VEL
LIN {X 0,Y 228.177,Z 281.4,A -85,B 0,C 180,E1 -20649.819,E2 -20649.819} C_VEL
LIN {X 0,Y 223.829,Z 273.678,A -85,B 0,C 180,E1 -20651.176,E2 -20651.176} C_VEL
LIN {X 0,Y 220.772,Z 268.493,A -85,B 0,C 180,E1 -20652.171,E2 -20652.171} C_VEL
LIN {X 0,Y 218.456,Z 264.606,A -85,B 0,C 180,E1 -20652.954,E2 -20652.954} C_VEL
LIN {X 0,Y 215.852,Z 260.144,A -85,B 0,C 180,E1 -20653.892,E2 -20653.892} C_VEL
LIN {X 0,Y 213.713,Z 252.864,A -85,B 0,C 180,E1 -20658.561,E2 -20658.561} C_VEL
LIN {X 0,Y 213.741,Z 252.852,A -85,B 0,C 180,E1 -20663.711,E2 -20663.711} C_VEL
LIN {X 0,Y 213.759,Z 252.857,A -85,B 0,C 180,E1 -20668.261,E2 -20668.261} C_VEL
LIN {X 0,Y 213.791,Z 252.854,A -85,B 0,C 180,E1 -20672.598,E2 -20672.598} C_VEL
LIN {X 0,Y 213.812,Z 252.853,A -85,B 0,C 180,E1 -20676.979,E2 -20676.979} C_VEL
LIN {X 0,Y 213.887,Z 252.835,A -85,B 0,C 180,E1 -20682.344,E2 -20682.344} C_VEL
LIN {X 0,Y 213.945,Z 252.829,A -85,B 0,C 180,E1 -20686.706,E2 -20686.706} C_VEL
LIN {X 0,Y 214.169,Z 252.806,A -85,B 0,C 180,E1 -20690.557,E2 -20690.557} C_VEL
LIN {X 0,Y 214.228,Z 252.787,A -85,B 0,C 180,E1 -20692.46,E2 -20692.46} C_VEL
LIN {X 0,Y 214.441,Z 252.758,A -85,B 0,C 180,E1 -20698.122,E2 -20698.122} C_VEL
LIN {X 0,Y 214.547,Z 252.758,A -85,B 0,C 180,E1 -20700,E2 -20700} C_VEL
LIN {X 0,Y 214.443,Z 252.765,A -85,B 0,C 180,E1 -20701.878,E2 -20701.878} C_VEL
LIN {X 0,Y 214.184,Z 252.793,A -85,B 0,C 180,E1 -20707.542,E2 -20707.542} C_VEL
LIN {X 0,Y 213.995,Z 252.828,A -85,B 0,C 180,E1 -20711.365,E2 -20711.365} C_VEL
LIN {X 0,Y 213.918,Z 252.835,A -85,B 0,C 180,E1 -20715.238,E2 -20715.238} C_VEL
LIN {X 0,Y 213.837,Z 252.839,A -85,B 0,C 180,E1 -20719.188,E2 -20719.188} C_VEL
LIN {X 0,Y 213.849,Z 252.836,A -85,B 0,C 180,E1 -20723.227,E2 -20723.227} C_VEL
LIN {X 0,Y 213.831,Z 252.842,A -85,B 0,C 180,E1 -20727.45,E2 -20727.45} C_VEL
LIN {X 0,Y 213.781,Z 252.857,A -85,B 0,C 180,E1 -20731.736,E2 -20731.736} C_VEL
LIN {X 0,Y 213.754,Z 252.853,A -85,B 0,C 180,E1 -20736.287,E2 -20736.287} C_VEL
LIN {X 0,Y 213.763,Z 252.854,A -85,B 0,C 180,E1 -20739.607,E2 -20739.607} C_VEL
LIN {X 0,Y 214.718,Z 255.64,A -85,B 0,C 180,E1 -20740.018,E2 -20740.018} C_VEL
LIN {X 0,Y 217.016,Z 258.264,A -85,B 0,C 180,E1 -20740.787,E2 -20740.787} C_VEL
LIN {X 0,Y 219.089,Z 261.545,A -85,B 0,C 180,E1 -20741.5,E2 -20741.5} C_VEL
LIN {X 0,Y 220.609,Z 263.541,A -85,B 0,C 180,E1 -20741.991,E2 -20741.991} C_VEL
LIN {X 0,Y 225.742,Z 271.228,A -85,B 0,C 180,E1 -20743.608,E2 -20743.608} C_VEL
LIN {X 0,Y 233.886,Z 285.959,A -85,B 0,C 180,E1 -20746.051,E2 -20746.051} C_VEL
LIN {X 0,Y 240.57,Z 300.093,A -85,B 0,C 180,E1 -20747.948,E2 -20747.948} C_VEL
LIN {X 0,Y 242.814,Z 305.423,A -85,B 0,C 180,E1 -20748.572,E2 -20748.572} C_VEL
LIN {X 0,Y 240.17,Z 359.244,A -85,B 0,C 180,E1 -20750.131,E2 -20750.131} C_VEL
LIN {X 0,Y 238.837,Z 372.42,A -85,B 0,C 180,E1 -20750.821,E2 -20750.821} C_VEL
LIN {X 0,Y 237.004,Z 384.539,A -85,B 0,C 180,E1 -20751.755,E2 -20751.755} C_VEL
LIN {X 0,Y 234.769,Z 395.937,A -85,B 0,C 180,E1 -20752.954,E2 -20752.954} C_VEL
LIN {X 0,Y 232.143,Z 406.343,A -85,B 0,C 180,E1 -20754.353,E2 -20754.353} C_VEL
LIN {X 0,Y 229.263,Z 416.652,A -85,B 0,C 180,E1 -20756.142,E2 -20756.142} C_VEL
LIN {X 0,Y 226.253,Z 425.828,A -85,B 0,C 180,E1 -20758.125,E2 -20758.125} C_VEL
LIN {X 0,Y 223.434,Z 433.859,A -85,B 0,C 180,E1 -20760.303,E2 -20760.303} C_VEL
LIN {X 0,Y 220.452,Z 441.81,A -85,B 0,C 180,E1 -20763.032,E2 -20763.032} C_VEL
LIN {X 0,Y 217.562,Z 448.844,A -85,B 0,C 180,E1 -20766.184,E2 -20766.184} C_VEL
LIN {X 0,Y 215.535,Z 453.59,A -85,B 0,C 180,E1 -20768.981,E2 -20768.981} C_VEL
LIN {X 0,Y 214.464,Z 456.139,A -85,B 0,C 180,E1 -20770.871,E2 -20770.871} C_VEL
LIN {X 0,Y 213.526,Z 458.176,A -85,B 0,C 180,E1 -20772.769,E2 -20772.769} C_VEL
LIN {X 0,Y 212.173,Z 461.002,A -85,B 0,C 180,E1 -20776.593,E2 -20776.593} C_VEL
LIN {X 0,Y 211.723,Z 461.78,A -85,B 0,C 180,E1 -20778.512,E2 -20778.512} C_VEL
LIN {X 0,Y 211.417,Z 462.124,A -85,B 0,C 180,E1 -20782.359,E2 -20782.359} C_VEL
LIN {X 0,Y 211.475,Z 461.205,A -85,B 0,C 180,E1 -20785.566,E2 -20785.566} C_VEL
LIN {X 0,Y 211.593,Z 459.675,A -85,B 0,C 180,E1 -20788.097,E2 -20788.097} C_VEL
LIN {X 0,Y 211.935,Z 457.076,A -85,B 0,C 180,E1 -20790.95,E2 -20790.95} C_VEL
LIN {X 0,Y 212.501,Z 453.482,A -85,B 0,C 180,E1 -20793.793,E2 -20793.793} C_VEL
LIN {X 0,Y 213.504,Z 448.784,A -85,B 0,C 180,E1 -20796.616,E2 -20796.616} C_VEL
LIN {X 0,Y 214.846,Z 442.847,A -85,B 0,C 180,E1 -20799.413,E2 -20799.413} C_VEL
LIN {X 0,Y 216.691,Z 435.452,A -85,B 0,C 180,E1 -20802.17,E2 -20802.17} C_VEL
LIN {X 0,Y 218.569,Z 427.908,A -85,B 0,C 180,E1 -20804.43,E2 -20804.43} C_VEL
LIN {X 0,Y 220.648,Z 418.782,A -85,B 0,C 180,E1 -20806.658,E2 -20806.658} C_VEL
LIN {X 0,Y 222.977,Z 407.606,A -85,B 0,C 180,E1 -20808.799,E2 -20808.799} C_VEL
LIN {X 0,Y 225.063,Z 395.802,A -85,B 0,C 180,E1 -20810.567,E2 -20810.567} C_VEL
LIN {X 0,Y 226.887,Z 383.547,A -85,B 0,C 180,E1 -20811.941,E2 -20811.941} C_VEL
LIN {X 0,Y 228.252,Z 370.67,A -85,B 0,C 180,E1 -20812.995,E2 -20812.995} C_VEL
LIN {X 0,Y 229.183,Z 357.91,A -85,B 0,C 180,E1 -20813.687,E2 -20813.687} C_VEL
LIN {X 0,Y 231.739,Z 292.962,A -85,B 0,C 180,E1 -20815.637,E2 -20815.637} C_VEL
LIN {X 0,Y 225.777,Z 277.299,A -85,B 0,C 180,E1 -20817.05,E2 -20817.05} C_VEL
LIN {X 0,Y 220.371,Z 265.413,A -85,B 0,C 180,E1 -20818.329,E2 -20818.329} C_VEL
LIN {X 0,Y 215.095,Z 256.13,A -85,B 0,C 180,E1 -20819.566,E2 -20819.566} C_VEL
LIN {X 0,Y 213.902,Z 253.482,A -85,B 0,C 180,E1 -20819.879,E2 -20819.879} C_VEL
LIN {X 0,Y 213.804,Z 252.853,A -85,B 0,C 180,E1 -20819.95,E2 -20819.95} C_VEL
LIN {X 0,Y 213.773,Z 252.857,A -85,B 0,C 180,E1 -20824.724,E2 -20824.724} C_VEL
LIN {X 0,Y 213.725,Z 252.862,A -85,B 0,C 180,E1 -20828.666,E2 -20828.666} C_VEL
LIN {X 0,Y 213.714,Z 252.862,A -85,B 0,C 180,E1 -20831.125,E2 -20831.125} C_VEL
LIN {X 0,Y 213.709,Z 252.862,A -85,B 0,C 180,E1 -20833.678,E2 -20833.678} C_VEL
LIN {X 0,Y 213.709,Z 252.865,A -85,B 0,C 180,E1 -20836.343,E2 -20836.343} C_VEL
LIN {X 0,Y 213.719,Z 252.863,A -85,B 0,C 180,E1 -20839.142,E2 -20839.142} C_VEL
LIN {X 0,Y 213.745,Z 252.859,A -85,B 0,C 180,E1 -20843.711,E2 -20843.711} C_VEL
LIN {X 0,Y 213.781,Z 252.834,A -85,B 0,C 180,E1 -20848.731,E2 -20848.731} C_VEL
LIN {X 0,Y 213.827,Z 252.851,A -85,B 0,C 180,E1 -20852.603,E2 -20852.603} C_VEL
LIN {X 0,Y 213.853,Z 252.817,A -85,B 0,C 180,E1 -20856.953,E2 -20856.953} C_VEL
LIN {X 0,Y 213.945,Z 252.833,A -85,B 0,C 180,E1 -20862.803,E2 -20862.803} C_VEL
LIN {X 0,Y 213.954,Z 252.812,A -85,B 0,C 180,E1 -20866.706,E2 -20866.706} C_VEL
LIN {X 0,Y 214.134,Z 252.785,A -85,B 0,C 180,E1 -20870.555,E2 -20870.555} C_VEL
LIN {X 0,Y 214.089,Z 252.814,A -85,B 0,C 180,E1 -20874.348,E2 -20874.348} C_VEL
LIN {X 0,Y 214.444,Z 252.762,A -85,B 0,C 180,E1 -20878.122,E2 -20878.122} C_VEL
LIN {X 0,Y 214.547,Z 252.757,A -85,B 0,C 180,E1 -20880,E2 -20880} C_VEL
LIN {X 0,Y 214.445,Z 252.77,A -85,B 0,C 180,E1 -20881.878,E2 -20881.878} C_VEL
LIN {X 0,Y 214.249,Z 252.796,A -85,B 0,C 180,E1 -20887.539,E2 -20887.539} C_VEL
LIN {X 0,Y 214.024,Z 252.81,A -85,B 0,C 180,E1 -20891.363,E2 -20891.363} C_VEL
LIN {X 0,Y 213.904,Z 252.839,A -85,B 0,C 180,E1 -20895.239,E2 -20895.239} C_VEL
LIN {X 0,Y 213.813,Z 252.841,A -85,B 0,C 180,E1 -20899.19,E2 -20899.19} C_VEL
LIN {X 0,Y 213.803,Z 252.849,A -85,B 0,C 180,E1 -20903.232,E2 -20903.232} C_VEL
LIN {X 0,Y 213.788,Z 252.854,A -85,B 0,C 180,E1 -20907.428,E2 -20907.428} C_VEL
LIN {X 0,Y 213.759,Z 252.855,A -85,B 0,C 180,E1 -20911.739,E2 -20911.739} C_VEL
LIN {X 0,Y 213.744,Z 252.858,A -85,B 0,C 180,E1 -20916.288,E2 -20916.288} C_VEL
LIN {X 0,Y 213.703,Z 252.864,A -85,B 0,C 180,E1 -20921.127,E2 -20921.127} C_VEL
LIN {X 0,Y 213.657,Z 252.864,A -85,B 0,C 180,E1 -20921.962,E2 -20921.962} C_VEL
LIN {X 0,Y 212.966,Z 252.957,A -85,B 0,C 180,E1 -20923.008,E2 -20923.008} C_VEL
LIN {X 0,Y 210.138,Z 253.307,A -85,B 0,C 180,E1 -20924.655,E2 -20924.655} C_VEL
LIN {X 0,Y 207.292,Z 253.664,A -85,B 0,C 180,E1 -20926.344,E2 -20926.344} C_VEL
LIN {X 0,Y 206.618,Z 253.739,A -85,B 0,C 180,E1 -20927.439,E2 -20927.439} C_VEL
LIN {X 0,Y 206.706,Z 253.844,A -85,B 0,C 180,E1 -20929.493,E2 -20929.493} C_VEL
LIN {X 0,Y 208.514,Z 260.835,A -85,B 0,C 180,E1 -20933.088,E2 -20933.088} C_VEL
LIN {X 0,Y 215.961,Z 277.059,A -85,B 0,C 180,E1 -20935.038,E2 -20935.038} C_VEL
LIN {X 0,Y 221.934,Z 292.231,A -85,B 0,C 180,E1 -20936.561,E2 -20936.561} C_VEL
LIN {X 0,Y 223.814,Z 305.993,A -85,B 0,C 180,E1 -20937.346,E2 -20937.346} C_VEL
LIN {X 0,Y 224.808,Z 315.923,A -85,B 0,C 180,E1 -20937.848,E2 -20937.848} C_VEL
LIN {X 0,Y 222.623,Z 369.523,A -85,B 0,C 180,E1 -20939.514,E2 -20939.514} C_VEL
LIN {X 0,Y 221.378,Z 382.998,A -85,B 0,C 180,E1 -20940.262,E2 -20940.262} C_VEL
LIN {X 0,Y 219.711,Z 395.697,A -85,B 0,C 180,E1 -20941.327,E2 -20941.327} C_VEL
LIN {X 0,Y 217.82,Z 406.966,A -85,B 0,C 180,E1 -20942.627,E2 -20942.627} C_VEL
LIN {X 0,Y 215.468,Z 418.634,A -85,B 0,C 180,E1 -20944.394,E2 -20944.394} C_VEL
LIN {X 0,Y 213.067,Z 429.128,A -85,B 0,C 180,E1 -20946.426,E2 -20946.426} C_VEL
LIN {X 0,Y 210.876,Z 438.8,A -85,B 0,C 180,E1 -20948.82,E2 -20948.82} C_VEL
LIN {X 0,Y 208.982,Z 447.008,A -85,B 0,C 180,E1 -20951.368,E2 -20951.368} C_VEL
LIN {X 0,Y 207.154,Z 454.46,A -85,B 0,C 180,E1 -20954.252,E2 -20954.252} C_VEL
LIN {X 0,Y 205.792,Z 460.435,A -85,B 0,C 180,E1 -20957.175,E2 -20957.175} C_VEL
LIN {X 0,Y 204.984,Z 465.151,A -85,B 0,C 180,E1 -20960.129,E2 -20960.129} C_VEL
LIN {X 0,Y 204.488,Z 468.738,A -85,B 0,C 180,E1 -20963.091,E2 -20963.091} C_VEL
LIN {X 0,Y 204.337,Z 471.306,A -85,B 0,C 180,E1 -20966.056,E2 -20966.056} C_VEL
LIN {X 0,Y 204.365,Z 472.509,A -85,B 0,C 180,E1 -20968.029,E2 -20968.029} C_VEL
LIN {X 0,Y 204.48,Z 473.266,A -85,B 0,C 180,E1 -20970,E2 -20970} C_VEL
LIN {X 0,Y 204.355,Z 473.615,A -85,B 0,C 180,E1 -20971.971,E2 -20971.971} C_VEL
LIN {X 0,Y 204.346,Z 473.563,A -85,B 0,C 180,E1 -20974.144,E2 -20974.144} C_VEL
LIN {X 0,Y 204.646,Z 472.323,A -85,B 0,C 180,E1 -20977.896,E2 -20977.896} C_VEL
LIN {X 0,Y 205.694,Z 469.426,A -85,B 0,C 180,E1 -20981.83,E2 -20981.83} C_VEL
LIN {X 0,Y 206.947,Z 466.13,A -85,B 0,C 180,E1 -20984.756,E2 -20984.756} C_VEL
LIN {X 0,Y 208.859,Z 461.783,A -85,B 0,C 180,E1 -20987.629,E2 -20987.629} C_VEL
LIN {X 0,Y 211.675,Z 455.238,A -85,B 0,C 180,E1 -20990.911,E2 -20990.911} C_VEL
LIN {X 0,Y 214.511,Z 448.068,A -85,B 0,C 180,E1 -20993.662,E2 -20993.662} C_VEL
LIN {X 0,Y 217.816,Z 439.178,A -85,B 0,C 180,E1 -20996.337,E2 -20996.337} C_VEL
LIN {X 0,Y 221.152,Z 430.063,A -85,B 0,C 180,E1 -20998.469,E2 -20998.469} C_VEL
LIN {X 0,Y 224.298,Z 419.97,A -85,B 0,C 180,E1 -21000.348,E2 -21000.348} C_VEL
LIN {X 0,Y 227.402,Z 408.774,A -85,B 0,C 180,E1 -21001.955,E2 -21001.955} C_VEL
LIN {X 0,Y 230.223,Z 396.207,A -85,B 0,C 180,E1 -21003.332,E2 -21003.332} C_VEL
LIN {X 0,Y 232.411,Z 383.232,A -85,B 0,C 180,E1 -21004.344,E2 -21004.344} C_VEL
LIN {X 0,Y 234.004,Z 370.073,A -85,B 0,C 180,E1 -21005.013,E2 -21005.013} C_VEL
LIN {X 0,Y 235.271,Z 346.326,A -85,B 0,C 180,E1 -21005.745,E2 -21005.745} C_VEL
LIN {X 0,Y 236.516,Z 320.114,A -85,B 0,C 180,E1 -21006.505,E2 -21006.505} C_VEL
LIN {X 0,Y 235.15,Z 310.882,A -85,B 0,C 180,E1 -21007.133,E2 -21007.133} C_VEL
LIN {X 0,Y 228.98,Z 296.536,A -85,B 0,C 180,E1 -21009.011,E2 -21009.011} C_VEL
LIN {X 0,Y 222.536,Z 283.504,A -85,B 0,C 180,E1 -21011.064,E2 -21011.064} C_VEL
LIN {X 0,Y 216.736,Z 273.356,A -85,B 0,C 180,E1 -21013.011,E2 -21013.011} C_VEL
LIN {X 0,Y 213.976,Z 268.833,A -85,B 0,C 180,E1 -21013.986,E2 -21013.986} C_VEL
LIN {X 0,Y 211.244,Z 264.495,A -85,B 0,C 180,E1 -21014.988,E2 -21014.988} C_VEL
LIN {X 0,Y 208.694,Z 260.303,A -85,B 0,C 180,E1 -21015.973,E2 -21015.973} C_VEL
LIN {X 0,Y 208.418,Z 259.542,A -85,B 0,C 180,E1 -21016.269,E2 -21016.269} C_VEL
LIN {X 0,Y 206.627,Z 253.745,A -85,B 0,C 180,E1 -21020.332,E2 -21020.332} C_VEL
LIN {X 0,Y 206.7,Z 253.737,A -85,B 0,C 180,E1 -21024.689,E2 -21024.689} C_VEL
LIN {X 0,Y 206.696,Z 253.732,A -85,B 0,C 180,E1 -21029.335,E2 -21029.335} C_VEL
LIN {X 0,Y 206.707,Z 253.728,A -85,B 0,C 180,E1 -21033.769,E2 -21033.769} C_VEL
LIN {X 0,Y 206.735,Z 253.725,A -85,B 0,C 180,E1 -21038.041,E2 -21038.041} C_VEL
LIN {X 0,Y 206.827,Z 253.715,A -85,B 0,C 180,E1 -21042.193,E2 -21042.193} C_VEL
LIN {X 0,Y 206.884,Z 253.713,A -85,B 0,C 180,E1 -21046.244,E2 -21046.244} C_VEL
LIN {X 0,Y 207.107,Z 253.686,A -85,B 0,C 180,E1 -21050.231,E2 -21050.231} C_VEL
LIN {X 0,Y 207.168,Z 253.667,A -85,B 0,C 180,E1 -21052.201,E2 -21052.201} C_VEL
LIN {X 0,Y 207.378,Z 253.637,A -85,B 0,C 180,E1 -21058.058,E2 -21058.058} C_VEL
LIN {X 0,Y 207.512,Z 253.634,A -85,B 0,C 180,E1 -21060,E2 -21060} C_VEL
LIN {X 0,Y 207.379,Z 253.644,A -85,B 0,C 180,E1 -21061.942,E2 -21061.942} C_VEL
LIN {X 0,Y 207.128,Z 253.67,A -85,B 0,C 180,E1 -21067.801,E2 -21067.801} C_VEL
LIN {X 0,Y 206.919,Z 253.706,A -85,B 0,C 180,E1 -21071.759,E2 -21071.759} C_VEL
LIN {X 0,Y 206.855,Z 253.717,A -85,B 0,C 180,E1 -21075.772,E2 -21075.772} C_VEL
LIN {X 0,Y 206.783,Z 253.723,A -85,B 0,C 180,E1 -21079.869,E2 -21079.869} C_VEL
LIN {X 0,Y 206.765,Z 253.726,A -85,B 0,C 180,E1 -21084.072,E2 -21084.072} C_VEL
LIN {X 0,Y 206.746,Z 253.731,A -85,B 0,C 180,E1 -21088.419,E2 -21088.419} C_VEL
LIN {X 0,Y 206.711,Z 253.731,A -85,B 0,C 180,E1 -21092.956,E2 -21092.956} C_VEL
LIN {X 0,Y 206.702,Z 253.737,A -85,B 0,C 180,E1 -21097.466,E2 -21097.466} C_VEL
LIN {X 0,Y 207.535,Z 256.285,A -85,B 0,C 180,E1 -21097.882,E2 -21097.882} C_VEL
LIN {X 0,Y 209.428,Z 258.498,A -85,B 0,C 180,E1 -21098.589,E2 -21098.589} C_VEL
LIN {X 0,Y 210.26,Z 259.417,A -85,B 0,C 180,E1 -21098.89,E2 -21098.89} C_VEL
LIN {X 0,Y 212.45,Z 262.757,A -85,B 0,C 180,E1 -21099.708,E2 -21099.708} C_VEL
LIN {X 0,Y 213.884,Z 264.75,A -85,B 0,C 180,E1 -21100.218,E2 -21100.218} C_VEL
LIN {X 0,Y 217.104,Z 269.316,A -85,B 0,C 180,E1 -21101.327,E2 -21101.327} C_VEL
LIN {X 0,Y 221.498,Z 275.905,A -85,B 0,C 180,E1 -21102.77,E2 -21102.77} C_VEL
LIN {X 0,Y 229.161,Z 289.957,A -85,B 0,C 180,E1 -21105.185,E2 -21105.185} C_VEL
LIN {X 0,Y 235.626,Z 303.853,A -85,B 0,C 180,E1 -21107.116,E2 -21107.116} C_VEL
LIN {X 0,Y 237.211,Z 307.588,A -85,B 0,C 180,E1 -21107.578,E2 -21107.578} C_VEL
LIN {X 0,Y 234.502,Z 359.6,A -85,B 0,C 180,E1 -21109.106,E2 -21109.106} C_VEL
LIN {X 0,Y 233.119,Z 372.724,A -85,B 0,C 180,E1 -21109.808,E2 -21109.808} C_VEL
LIN {X 0,Y 231.223,Z 384.816,A -85,B 0,C 180,E1 -21110.758,E2 -21110.758} C_VEL
LIN {X 0,Y 228.7,Z 396.988,A -85,B 0,C 180,E1 -21112.077,E2 -21112.077} C_VEL
LIN {X 0,Y 225.975,Z 407.236,A -85,B 0,C 180,E1 -21113.501,E2 -21113.501} C_VEL
LIN {X 0,Y 222.87,Z 417.854,A -85,B 0,C 180,E1 -21115.416,E2 -21115.416} C_VEL
LIN {X 0,Y 219.544,Z 427.389,A -85,B 0,C 180,E1 -21117.575,E2 -21117.575} C_VEL
LIN {X 0,Y 216.66,Z 435.17,A -85,B 0,C 180,E1 -21119.815,E2 -21119.815} C_VEL
LIN {X 0,Y 213.439,Z 443.187,A -85,B 0,C 180,E1 -21122.754,E2 -21122.754} C_VEL
LIN {X 0,Y 211.005,Z 448.83,A -85,B 0,C 180,E1 -21125.396,E2 -21125.396} C_VEL
LIN {X 0,Y 208.806,Z 453.621,A -85,B 0,C 180,E1 -21128.27,E2 -21128.27} C_VEL
LIN {X 0,Y 207.15,Z 457.278,A -85,B 0,C 180,E1 -21131.197,E2 -21131.197} C_VEL
LIN {X 0,Y 205.822,Z 459.905,A -85,B 0,C 180,E1 -21134.147,E2 -21134.147} C_VEL
LIN {X 0,Y 205.186,Z 461.134,A -85,B 0,C 180,E1 -21136.127,E2 -21136.127} C_VEL
LIN {X 0,Y 204.693,Z 461.95,A -85,B 0,C 180,E1 -21138.112,E2 -21138.112} C_VEL
LIN {X 0,Y 204.342,Z 462.331,A -85,B 0,C 180,E1 -21142.092,E2 -21142.092} C_VEL
LIN {X 0,Y 204.386,Z 461.326,A -85,B 0,C 180,E1 -21145.712,E2 -21145.712} C_VEL
LIN {X 0,Y 204.485,Z 459.957,A -85,B 0,C 180,E1 -21148.03,E2 -21148.03} C_VEL
LIN {X 0,Y 204.862,Z 457.396,A -85,B 0,C 180,E1 -21150.983,E2 -21150.983} C_VEL
LIN {X 0,Y 205.442,Z 453.844,A -85,B 0,C 180,E1 -21153.923,E2 -21153.923} C_VEL
LIN {X 0,Y 206.474,Z 449.19,A -85,B 0,C 180,E1 -21156.842,E2 -21156.842} C_VEL
LIN {X 0,Y 207.872,Z 443.302,A -85,B 0,C 180,E1 -21159.732,E2 -21159.732} C_VEL
LIN {X 0,Y 209.787,Z 435.961,A -85,B 0,C 180,E1 -21162.577,E2 -21162.577} C_VEL
LIN {X 0,Y 212.097,Z 426.84,A -85,B 0,C 180,E1 -21165.372,E2 -21165.372} C_VEL
LIN {X 0,Y 214.614,Z 416.296,A -85,B 0,C 180,E1 -21167.879,E2 -21167.879} C_VEL
LIN {X 0,Y 216.984,Z 405.074,A -85,B 0,C 180,E1 -21169.972,E2 -21169.972} C_VEL
LIN {X 0,Y 219.046,Z 393.36,A -85,B 0,C 180,E1 -21171.652,E2 -21171.652} C_VEL
LIN {X 0,Y 220.786,Z 381.422,A -85,B 0,C 180,E1 -21172.951,E2 -21172.951} C_VEL
LIN {X 0,Y 222.155,Z 368.364,A -85,B 0,C 180,E1 -21173.974,E2 -21173.974} C_VEL
LIN {X 0,Y 223.029,Z 355.719,A -85,B 0,C 180,E1 -21174.599,E2 -21174.599} C_VEL
LIN {X 0,Y 225.516,Z 294.573,A -85,B 0,C 180,E1 -21176.464,E2 -21176.464} C_VEL
LIN {X 0,Y 219.181,Z 278.207,A -85,B 0,C 180,E1 -21178.038,E2 -21178.038} C_VEL
LIN {X 0,Y 215.005,Z 269.154,A -85,B 0,C 180,E1 -21179.074,E2 -21179.074} C_VEL
LIN {X 0,Y 208.4,Z 257.436,A -85,B 0,C 180,E1 -21180.718,E2 -21180.718} C_VEL
LIN {X 0,Y 206.919,Z 254.696,A -85,B 0,C 180,E1 -21181.11,E2 -21181.11} C_VEL
LIN {X 0,Y 206.726,Z 253.735,A -85,B 0,C 180,E1 -21181.224,E2 -21181.224} C_VEL
LIN {X 0,Y 206.701,Z 253.736,A -85,B 0,C 180,E1 -21185.311,E2 -21185.311} C_VEL
LIN {X 0,Y 206.663,Z 253.741,A -85,B 0,C 180,E1 -21190.251,E2 -21190.251} C_VEL
LIN {X 0,Y 206.636,Z 253.746,A -85,B 0,C 180,E1 -21194.418,E2 -21194.418} C_VEL
LIN {X 0,Y 206.644,Z 253.744,A -85,B 0,C 180,E1 -21198.437,E2 -21198.437} C_VEL
LIN {X 0,Y 206.681,Z 253.737,A -85,B 0,C 180,E1 -21202.26,E2 -21202.26} C_VEL
LIN {X 0,Y 206.7,Z 253.713,A -85,B 0,C 180,E1 -21207.042,E2 -21207.042} C_VEL
LIN {X 0,Y 206.765,Z 253.728,A -85,B 0,C 180,E1 -21212.097,E2 -21212.097} C_VEL
LIN {X 0,Y 206.786,Z 253.698,A -85,B 0,C 180,E1 -21216.584,E2 -21216.584} C_VEL
LIN {X 0,Y 206.875,Z 253.71,A -85,B 0,C 180,E1 -21222.196,E2 -21222.196} C_VEL
LIN {X 0,Y 206.896,Z 253.694,A -85,B 0,C 180,E1 -21226.244,E2 -21226.244} C_VEL
LIN {X 0,Y 207.079,Z 253.66,A -85,B 0,C 180,E1 -21230.23,E2 -21230.23} C_VEL
LIN {X 0,Y 207.05,Z 253.689,A -85,B 0,C 180,E1 -21234.155,E2 -21234.155} C_VEL
LIN {X 0,Y 207.38,Z 253.641,A -85,B 0,C 180,E1 -21238.058,E2 -21238.058} C_VEL
LIN {X 0,Y 207.512,Z 253.633,A -85,B 0,C 180,E1 -21240,E2 -21240} C_VEL
LIN {X 0,Y 207.381,Z 253.65,A -85,B 0,C 180,E1 -21241.942,E2 -21241.942} C_VEL
LIN {X 0,Y 207.189,Z 253.675,A -85,B 0,C 180,E1 -21247.798,E2 -21247.798} C_VEL
LIN {X 0,Y 206.941,Z 253.693,A -85,B 0,C 180,E1 -21251.757,E2 -21251.757} C_VEL
LIN {X 0,Y 206.832,Z 253.719,A -85,B 0,C 180,E1 -21255.773,E2 -21255.773} C_VEL
LIN {X 0,Y 206.749,Z 253.724,A -85,B 0,C 180,E1 -21259.872,E2 -21259.872} C_VEL
LIN {X 0,Y 206.738,Z 253.726,A -85,B 0,C 180,E1 -21264.075,E2 -21264.075} C_VEL
LIN {X 0,Y 206.689,Z 253.739,A -85,B 0,C 180,E1 -21268.427,E2 -21268.427} C_VEL
LIN {X 0,Y 206.695,Z 253.738,A -85,B 0,C 180,E1 -21272.958,E2 -21272.958} C_VEL
LIN {X 0,Y 206.674,Z 253.74,A -85,B 0,C 180,E1 -21277.741,E2 -21277.741} C_VEL
LIN {X 0,Y 206.619,Z 253.744,A -85,B 0,C 180,E1 -21281.947,E2 -21281.947} C_VEL
LIN {X 0,Y 206.632,Z 253.743,A -85,B 0,C 180,E1 -21285.582,E2 -21285.582} C_VEL
LIN {X 0,Y 206.618,Z 253.739,A -85,B 0,C 180,E1 -21287.439,E2 -21287.439} C_VEL
LIN {X 0,Y 206.09,Z 254.328,A -85,B 0,C 180,E1 -21288.592,E2 -21288.592} C_VEL
LIN {X 0,Y 204.543,Z 256.539,A -85,B 0,C 180,E1 -21290.003,E2 -21290.003} C_VEL
LIN {X 0,Y 203.202,Z 259.918,A -85,B 0,C 180,E1 -21291.224,E2 -21291.224} C_VEL
LIN {X 0,Y 203.034,Z 263.39,A -85,B 0,C 180,E1 -21292.027,E2 -21292.027} C_VEL
LIN {X 0,Y 203.574,Z 265.441,A -85,B 0,C 180,E1 -21292.339,E2 -21292.339} C_VEL
LIN {X 0,Y 210.351,Z 280.122,A -85,B 0,C 180,E1 -21294.198,E2 -21294.198} C_VEL
LIN {X 0,Y 216.232,Z 295.25,A -85,B 0,C 180,E1 -21295.78,E2 -21295.78} C_VEL
LIN {X 0,Y 218.644,Z 316.136,A -85,B 0,C 180,E1 -21296.946,E2 -21296.946} C_VEL
LIN {X 0,Y 216.29,Z 370.184,A -85,B 0,C 180,E1 -21298.675,E2 -21298.675} C_VEL
LIN {X 0,Y 215.04,Z 383.186,A -85,B 0,C 180,E1 -21299.428,E2 -21299.428} C_VEL
LIN {X 0,Y 213.31,Z 395.777,A -85,B 0,C 180,E1 -21300.518,E2 -21300.518} C_VEL
LIN {X 0,Y 211.216,Z 407.768,A -85,B 0,C 180,E1 -21301.966,E2 -21301.966} C_VEL
LIN {X 0,Y 208.767,Z 419.252,A -85,B 0,C 180,E1 -21303.778,E2 -21303.778} C_VEL
LIN {X 0,Y 206.28,Z 429.598,A -85,B 0,C 180,E1 -21305.868,E2 -21305.868} C_VEL
LIN {X 0,Y 204.135,Z 438.687,A -85,B 0,C 180,E1 -21308.211,E2 -21308.211} C_VEL
LIN {X 0,Y 202.254,Z 446.558,A -85,B 0,C 180,E1 -21310.725,E2 -21310.725} C_VEL
LIN {X 0,Y 200.289,Z 454.052,A -85,B 0,C 180,E1 -21313.697,E2 -21313.697} C_VEL
LIN {X 0,Y 198.828,Z 460.067,A -85,B 0,C 180,E1 -21316.717,E2 -21316.717} C_VEL
LIN {X 0,Y 197.959,Z 464.82,A -85,B 0,C 180,E1 -21319.775,E2 -21319.775} C_VEL
LIN {X 0,Y 197.433,Z 468.442,A -85,B 0,C 180,E1 -21322.843,E2 -21322.843} C_VEL
LIN {X 0,Y 197.248,Z 471.154,A -85,B 0,C 180,E1 -21326.071,E2 -21326.071} C_VEL
LIN {X 0,Y 197.27,Z 472.263,A -85,B 0,C 180,E1 -21327.958,E2 -21327.958} C_VEL
LIN {X 0,Y 197.38,Z 473.047,A -85,B 0,C 180,E1 -21330,E2 -21330} C_VEL
LIN {X 0,Y 197.243,Z 473.407,A -85,B 0,C 180,E1 -21333.909,E2 -21333.909} C_VEL
LIN {X 0,Y 197.342,Z 472.988,A -85,B 0,C 180,E1 -21336.133,E2 -21336.133} C_VEL
LIN {X 0,Y 197.597,Z 472.178,A -85,B 0,C 180,E1 -21338.179,E2 -21338.179} C_VEL
LIN {X 0,Y 198.71,Z 469.313,A -85,B 0,C 180,E1 -21342.252,E2 -21342.252} C_VEL
LIN {X 0,Y 200.07,Z 466.049,A -85,B 0,C 180,E1 -21345.275,E2 -21345.275} C_VEL
LIN {X 0,Y 202.099,Z 461.737,A -85,B 0,C 180,E1 -21348.239,E2 -21348.239} C_VEL
LIN {X 0,Y 205.061,Z 455.24,A -85,B 0,C 180,E1 -21351.619,E2 -21351.619} C_VEL
LIN {X 0,Y 208.012,Z 448.124,A -85,B 0,C 180,E1 -21354.449,E2 -21354.449} C_VEL
LIN {X 0,Y 211.48,Z 439.285,A -85,B 0,C 180,E1 -21357.19,E2 -21357.19} C_VEL
LIN {X 0,Y 214.944,Z 430.231,A -85,B 0,C 180,E1 -21359.37,E2 -21359.37} C_VEL
LIN {X 0,Y 218.219,Z 420.253,A -85,B 0,C 180,E1 -21361.287,E2 -21361.287} C_VEL
LIN {X 0,Y 221.44,Z 409.167,A -85,B 0,C 180,E1 -21362.923,E2 -21362.923} C_VEL
LIN {X 0,Y 224.341,Z 396.755,A -85,B 0,C 180,E1 -21364.325,E2 -21364.325} C_VEL
LIN {X 0,Y 226.632,Z 384.17,A -85,B 0,C 180,E1 -21365.348,E2 -21365.348} C_VEL
LIN {X 0,Y 228.244,Z 371.507,A -85,B 0,C 180,E1 -21366.037,E2 -21366.037} C_VEL
LIN {X 0,Y 229.399,Z 354.707,A -85,B 0,C 180,E1 -21366.578,E2 -21366.578} C_VEL
LIN {X 0,Y 231.04,Z 321.588,A -85,B 0,C 180,E1 -21367.555,E2 -21367.555} C_VEL
LIN {X 0,Y 229.786,Z 313.39,A -85,B 0,C 180,E1 -21368.149,E2 -21368.149} C_VEL
LIN {X 0,Y 223.718,Z 299.244,A -85,B 0,C 180,E1 -21370.099,E2 -21370.099} C_VEL
LIN {X 0,Y 217.897,Z 287.396,A -85,B 0,C 180,E1 -21372.059,E2 -21372.059} C_VEL
LIN {X 0,Y 212.633,Z 278.063,A -85,B 0,C 180,E1 -21373.924,E2 -21373.924} C_VEL
LIN {X 0,Y 209.707,Z 273.195,A -85,B 0,C 180,E1 -21375.015,E2 -21375.015} C_VEL
LIN {X 0,Y 207.506,Z 269.652,A -85,B 0,C 180,E1 -21375.865,E2 -21375.865} C_VEL
LIN {X 0,Y 204.102,Z 264.336,A -85,B 0,C 180,E1 -21377.238,E2 -21377.238} C_VEL
LIN {X 0,Y 201.352,Z 260.132,A -85,B 0,C 180,E1 -21378.406,E2 -21378.406} C_VEL
LIN {X 0,Y 201.045,Z 259.28,A -85,B 0,C 180,E1 -21378.714,E2 -21378.714} C_VEL
LIN {X 0,Y 199.634,Z 254.611,A -85,B 0,C 180,E1 -21382.289,E2 -21382.289} C_VEL
LIN {X 0,Y 199.686,Z 254.608,A -85,B 0,C 180,E1 -21388.134,E2 -21388.134} C_VEL
LIN {X 0,Y 199.645,Z 254.616,A -85,B 0,C 180,E1 -21392.766,E2 -21392.766} C_VEL
LIN {X 0,Y 199.709,Z 254.606,A -85,B 0,C 180,E1 -21397.226,E2 -21397.226} C_VEL
LIN {X 0,Y 199.751,Z 254.6,A -85,B 0,C 180,E1 -21401.798,E2 -21401.798} C_VEL
LIN {X 0,Y 199.821,Z 254.595,A -85,B 0,C 180,E1 -21405.747,E2 -21405.747} C_VEL
LIN {X 0,Y 200.072,Z 254.56,A -85,B 0,C 180,E1 -21409.884,E2 -21409.884} C_VEL
LIN {X 0,Y 200.03,Z 254.557,A -85,B 0,C 180,E1 -21413.95,E2 -21413.95} C_VEL
LIN {X 0,Y 200.317,Z 254.517,A -85,B 0,C 180,E1 -21417.99,E2 -21417.99} C_VEL
LIN {X 0,Y 200.477,Z 254.51,A -85,B 0,C 180,E1 -21420,E2 -21420} C_VEL
LIN {X 0,Y 200.017,Z 254.558,A -85,B 0,C 180,E1 -21424.03,E2 -21424.03} C_VEL
LIN {X 0,Y 200.076,Z 254.548,A -85,B 0,C 180,E1 -21428.077,E2 -21428.077} C_VEL
LIN {X 0,Y 199.869,Z 254.58,A -85,B 0,C 180,E1 -21432.18,E2 -21432.18} C_VEL
LIN {X 0,Y 199.796,Z 254.595,A -85,B 0,C 180,E1 -21436.344,E2 -21436.344} C_VEL
LIN {X 0,Y 199.7,Z 254.607,A -85,B 0,C 180,E1 -21440.606,E2 -21440.606} C_VEL
LIN {X 0,Y 199.675,Z 254.609,A -85,B 0,C 180,E1 -21444.984,E2 -21444.984} C_VEL
LIN {X 0,Y 199.677,Z 254.605,A -85,B 0,C 180,E1 -21449.522,E2 -21449.522} C_VEL
LIN {X 0,Y 199.666,Z 254.612,A -85,B 0,C 180,E1 -21452.353,E2 -21452.353} C_VEL
LIN {X 0,Y 199.682,Z 254.625,A -85,B 0,C 180,E1 -21455.112,E2 -21455.112} C_VEL
LIN {X 0,Y 200.574,Z 257.3,A -85,B 0,C 180,E1 -21455.586,E2 -21455.586} C_VEL
LIN {X 0,Y 202.642,Z 259.545,A -85,B 0,C 180,E1 -21456.437,E2 -21456.437} C_VEL
LIN {X 0,Y 203.287,Z 260.114,A -85,B 0,C 180,E1 -21456.688,E2 -21456.688} C_VEL
LIN {X 0,Y 205.237,Z 263.332,A -85,B 0,C 180,E1 -21457.51,E2 -21457.51} C_VEL
LIN {X 0,Y 206.96,Z 265.363,A -85,B 0,C 180,E1 -21458.17,E2 -21458.17} C_VEL
LIN {X 0,Y 213.736,Z 275.151,A -85,B 0,C 180,E1 -21460.675,E2 -21460.675} C_VEL
LIN {X 0,Y 217.971,Z 281.837,A -85,B 0,C 180,E1 -21462.133,E2 -21462.133} C_VEL
LIN {X 0,Y 225.026,Z 295.085,A -85,B 0,C 180,E1 -21464.456,E2 -21464.456} C_VEL
LIN {X 0,Y 231.173,Z 308.616,A -85,B 0,C 180,E1 -21466.381,E2 -21466.381} C_VEL
LIN {X 0,Y 231.637,Z 309.663,A -85,B 0,C 180,E1 -21466.521,E2 -21466.521} C_VEL
LIN {X 0,Y 228.986,Z 359.207,A -85,B 0,C 180,E1 -21467.999,E2 -21467.999} C_VEL
LIN {X 0,Y 227.589,Z 372.194,A -85,B 0,C 180,E1 -21468.688,E2 -21468.688} C_VEL
LIN {X 0,Y 225.503,Z 385.095,A -85,B 0,C 180,E1 -21469.707,E2 -21469.707} C_VEL
LIN {X 0,Y 223.092,Z 396.444,A -85,B 0,C 180,E1 -21470.946,E2 -21470.946} C_VEL
LIN {X 0,Y 220.261,Z 406.827,A -85,B 0,C 180,E1 -21472.394,E2 -21472.394} C_VEL
LIN {X 0,Y 216.972,Z 417.548,A -85,B 0,C 180,E1 -21474.335,E2 -21474.335} C_VEL
LIN {X 0,Y 213.539,Z 427.181,A -85,B 0,C 180,E1 -21476.545,E2 -21476.545} C_VEL
LIN {X 0,Y 210.444,Z 435.042,A -85,B 0,C 180,E1 -21478.826,E2 -21478.826} C_VEL
LIN {X 0,Y 207.218,Z 442.69,A -85,B 0,C 180,E1 -21481.652,E2 -21481.652} C_VEL
LIN {X 0,Y 204.477,Z 448.815,A -85,B 0,C 180,E1 -21484.556,E2 -21484.556} C_VEL
LIN {X 0,Y 202.123,Z 453.652,A -85,B 0,C 180,E1 -21487.512,E2 -21487.512} C_VEL
LIN {X 0,Y 200.328,Z 457.352,A -85,B 0,C 180,E1 -21490.532,E2 -21490.532} C_VEL
LIN {X 0,Y 198.92,Z 460.018,A -85,B 0,C 180,E1 -21493.582,E2 -21493.582} C_VEL
LIN {X 0,Y 198.22,Z 461.267,A -85,B 0,C 180,E1 -21495.63,E2 -21495.63} C_VEL
LIN {X 0,Y 197.673,Z 462.114,A -85,B 0,C 180,E1 -21497.683,E2 -21497.683} C_VEL
LIN {X 0,Y 197.26,Z 462.538,A -85,B 0,C 180,E1 -21501.807,E2 -21501.807} C_VEL
LIN {X 0,Y 197.269,Z 462.173,A -85,B 0,C 180,E1 -21503.864,E2 -21503.864} C_VEL
LIN {X 0,Y 197.307,Z 461.423,A -85,B 0,C 180,E1 -21505.915,E2 -21505.915} C_VEL
LIN {X 0,Y 197.382,Z 460.238,A -85,B 0,C 180,E1 -21507.959,E2 -21507.959} C_VEL
LIN {X 0,Y 197.617,Z 458.65,A -85,B 0,C 180,E1 -21510,E2 -21510} C_VEL
LIN {X 0,Y 198.15,Z 455.472,A -85,B 0,C 180,E1 -21513.05,E2 -21513.05} C_VEL
LIN {X 0,Y 199.037,Z 451.243,A -85,B 0,C 180,E1 -21516.081,E2 -21516.081} C_VEL
LIN {X 0,Y 200.706,Z 444.832,A -85,B 0,C 180,E1 -21519.574,E2 -21519.574} C_VEL
LIN {X 0,Y 202.525,Z 437.817,A -85,B 0,C 180,E1 -21522.526,E2 -21522.526} C_VEL
LIN {X 0,Y 204.902,Z 429.053,A -85,B 0,C 180,E1 -21525.416,E2 -21525.416} C_VEL
LIN {X 0,Y 207.423,Z 419.1,A -85,B 0,C 180,E1 -21528.01,E2 -21528.01} C_VEL
LIN {X 0,Y 209.759,Z 408.672,A -85,B 0,C 180,E1 -21530.137,E2 -21530.137} C_VEL
LIN {X 0,Y 211.922,Z 397.653,A -85,B 0,C 180,E1 -21531.906,E2 -21531.906} C_VEL
LIN {X 0,Y 213.871,Z 385.953,A -85,B 0,C 180,E1 -21533.352,E2 -21533.352} C_VEL
LIN {X 0,Y 215.422,Z 373.123,A -85,B 0,C 180,E1 -21534.516,E2 -21534.516} C_VEL
LIN {X 0,Y 216.542,Z 359.866,A -85,B 0,C 180,E1 -21535.314,E2 -21535.314} C_VEL
LIN {X 0,Y 218.774,Z 311.426,A -85,B 0,C 180,E1 -21536.856,E2 -21536.856} C_VEL
LIN {X 0,Y 219.333,Z 296.251,A -85,B 0,C 180,E1 -21537.336,E2 -21537.336} C_VEL
LIN {X 0,Y 213.487,Z 281.173,A -85,B 0,C 180,E1 -21538.864,E2 -21538.864} C_VEL
LIN {X 0,Y 209.537,Z 272.597,A -85,B 0,C 180,E1 -21539.895,E2 -21539.895} C_VEL
LIN {X 0,Y 203.218,Z 261.51,A -85,B 0,C 180,E1 -21541.543,E2 -21541.543} C_VEL
LIN {X 0,Y 201.28,Z 258.319,A -85,B 0,C 180,E1 -21542.067,E2 -21542.067} C_VEL
LIN {X 0,Y 199.904,Z 255.77,A -85,B 0,C 180,E1 -21542.46,E2 -21542.46} C_VEL
LIN {X 0,Y 199.654,Z 254.616,A -85,B 0,C 180,E1 -21542.603,E2 -21542.603} C_VEL
LIN {X 0,Y 199.625,Z 254.618,A -85,B 0,C 180,E1 -21546.763,E2 -21546.763} C_VEL
LIN {X 0,Y 199.61,Z 254.619,A -85,B 0,C 180,E1 -21549.328,E2 -21549.328} C_VEL
LIN {X 0,Y 199.577,Z 254.624,A -85,B 0,C 180,E1 -21552.31,E2 -21552.31} C_VEL
LIN {X 0,Y 199.583,Z 254.623,A -85,B 0,C 180,E1 -21555.229,E2 -21555.229} C_VEL
LIN {X 0,Y 199.582,Z 254.623,A -85,B 0,C 180,E1 -21558.005,E2 -21558.005} C_VEL
LIN {X 0,Y 199.612,Z 254.617,A -85,B 0,C 180,E1 -21560.767,E2 -21560.767} C_VEL
LIN {X 0,Y 199.613,Z 254.608,A -85,B 0,C 180,E1 -21565.713,E2 -21565.713} C_VEL
LIN {X 0,Y 199.694,Z 254.583,A -85,B 0,C 180,E1 -21568.135,E2 -21568.135} C_VEL
LIN {X 0,Y 199.687,Z 254.61,A -85,B 0,C 180,E1 -21572.771,E2 -21572.771} C_VEL
LIN {X 0,Y 199.739,Z 254.57,A -85,B 0,C 180,E1 -21577.229,E2 -21577.229} C_VEL
LIN {X 0,Y 199.798,Z 254.591,A -85,B 0,C 180,E1 -21581.757,E2 -21581.757} C_VEL
LIN {X 0,Y 199.837,Z 254.578,A -85,B 0,C 180,E1 -21585.748,E2 -21585.748} C_VEL
LIN {X 0,Y 200.023,Z 254.534,A -85,B 0,C 180,E1 -21589.882,E2 -21589.882} C_VEL
LIN {X 0,Y 200.012,Z 254.565,A -85,B 0,C 180,E1 -21593.949,E2 -21593.949} C_VEL
LIN {X 0,Y 200.319,Z 254.52,A -85,B 0,C 180,E1 -21597.989,E2 -21597.989} C_VEL
LIN {X 0,Y 200.477,Z 254.509,A -85,B 0,C 180,E1 -21600,E2 -21600} C_VEL
LIN {X 0,Y 200.028,Z 254.559,A -85,B 0,C 180,E1 -21604.029,E2 -21604.029} C_VEL
LIN {X 0,Y 200.133,Z 254.555,A -85,B 0,C 180,E1 -21608.075,E2 -21608.075} C_VEL
LIN {X 0,Y 200.069,Z 254.549,A -85,B 0,C 180,E1 -21610.397,E2 -21610.397} C_VEL
LIN {X 0,Y 199.768,Z 254.598,A -85,B 0,C 180,E1 -21616.346,E2 -21616.346} C_VEL
LIN {X 0,Y 199.672,Z 254.609,A -85,B 0,C 180,E1 -21620.608,E2 -21620.608} C_VEL
LIN {X 0,Y 199.651,Z 254.605,A -85,B 0,C 180,E1 -21624.987,E2 -21624.987} C_VEL
LIN {X 0,Y 199.609,Z 254.616,A -85,B 0,C 180,E1 -21629.533,E2 -21629.533} C_VEL
LIN {X 0,Y 199.666,Z 254.613,A -85,B 0,C 180,E1 -21632.353,E2 -21632.353} C_VEL
LIN {X 0,Y 199.62,Z 254.62,A -85,B 0,C 180,E1 -21636.764,E2 -21636.764} C_VEL
LIN {X 0,Y 199.597,Z 254.618,A -85,B 0,C 180,E1 -21639.331,E2 -21639.331} C_VEL
LIN {X 0,Y 199.568,Z 254.622,A -85,B 0,C 180,E1 -21642.308,E2 -21642.308} C_VEL
LIN {X 0,Y 199.578,Z 254.621,A -85,B 0,C 180,E1 -21645.228,E2 -21645.228} C_VEL
LIN {X 0,Y 199.628,Z 254.689,A -85,B 0,C 180,E1 -21648.453,E2 -21648.453} C_VEL
LIN {X 0,Y 201.21,Z 260.652,A -85,B 0,C 180,E1 -21651.665,E2 -21651.665} C_VEL
LIN {X 0,Y 203.574,Z 265.441,A -85,B 0,C 180,E1 -21652.339,E2 -21652.339} C_VEL
LIN {X 0,Y 205.193,Z 270.811,A -85,B 0,C 180,E1 -21652.875,E2 -21652.875} C_VEL
LIN {X 0,Y 207.676,Z 288.037,A -85,B 0,C 180,E1 -21654.04,E2 -21654.04} C_VEL
LIN {X 0,Y 208.965,Z 293.608,A -85,B 0,C 180,E1 -21654.493,E2 -21654.493} C_VEL
LIN {X 0,Y 209.568,Z 295.384,A -85,B 0,C 180,E1 -21654.669,E2 -21654.669} C_VEL
LIN {X 0,Y 210.484,Z 298.445,A -85,B 0,C 180,E1 -21654.949,E2 -21654.949} C_VEL
LIN {X 0,Y 212.515,Z 316.817,A -85,B 0,C 180,E1 -21656.006,E2 -21656.006} C_VEL
LIN {X 0,Y 210.161,Z 369.423,A -85,B 0,C 180,E1 -21657.723,E2 -21657.723} C_VEL
LIN {X 0,Y 208.842,Z 382.608,A -85,B 0,C 180,E1 -21658.489,E2 -21658.489} C_VEL
LIN {X 0,Y 207.145,Z 394.741,A -85,B 0,C 180,E1 -21659.549,E2 -21659.549} C_VEL
LIN {X 0,Y 204.937,Z 406.974,A -85,B 0,C 180,E1 -21661.027,E2 -21661.027} C_VEL
LIN {X 0,Y 202.419,Z 418.571,A -85,B 0,C 180,E1 -21662.89,E2 -21662.89} C_VEL
LIN {X 0,Y 199.822,Z 429.008,A -85,B 0,C 180,E1 -21665.036,E2 -21665.036} C_VEL
LIN {X 0,Y 197.415,Z 438.573,A -85,B 0,C 180,E1 -21667.561,E2 -21667.561} C_VEL
LIN {X 0,Y 195.551,Z 446.107,A -85,B 0,C 180,E1 -21670.036,E2 -21670.036} C_VEL
LIN {X 0,Y 193.458,Z 453.645,A -85,B 0,C 180,E1 -21673.105,E2 -21673.105} C_VEL
LIN {X 0,Y 191.887,Z 459.699,A -85,B 0,C 180,E1 -21676.228,E2 -21676.228} C_VEL
LIN {X 0,Y 190.952,Z 464.489,A -85,B 0,C 180,E1 -21679.396,E2 -21679.396} C_VEL
LIN {X 0,Y 190.363,Z 468.145,A -85,B 0,C 180,E1 -21682.576,E2 -21682.576} C_VEL
LIN {X 0,Y 190.16,Z 471.124,A -85,B 0,C 180,E1 -21686.266,E2 -21686.266} C_VEL
LIN {X 0,Y 190.282,Z 472.828,A -85,B 0,C 180,E1 -21690,E2 -21690} C_VEL
LIN {X 0,Y 190.134,Z 473.254,A -85,B 0,C 180,E1 -21693.614,E2 -21693.614} C_VEL
LIN {X 0,Y 190.28,Z 472.814,A -85,B 0,C 180,E1 -21696.362,E2 -21696.362} C_VEL
LIN {X 0,Y 190.547,Z 472.031,A -85,B 0,C 180,E1 -21698.484,E2 -21698.484} C_VEL
LIN {X 0,Y 191.749,Z 469.199,A -85,B 0,C 180,E1 -21702.704,E2 -21702.704} C_VEL
LIN {X 0,Y 193.219,Z 465.969,A -85,B 0,C 180,E1 -21705.831,E2 -21705.831} C_VEL
LIN {X 0,Y 195.366,Z 461.691,A -85,B 0,C 180,E1 -21708.891,E2 -21708.891} C_VEL
LIN {X 0,Y 198.475,Z 455.236,A -85,B 0,C 180,E1 -21712.374,E2 -21712.374} C_VEL
LIN {X 0,Y 201.545,Z 448.182,A -85,B 0,C 180,E1 -21715.288,E2 -21715.288} C_VEL
LIN {X 0,Y 205.18,Z 439.395,A -85,B 0,C 180,E1 -21718.098,E2 -21718.098} C_VEL
LIN {X 0,Y 209.12,Z 429.427,A -85,B 0,C 180,E1 -21720.552,E2 -21720.552} C_VEL
LIN {X 0,Y 212.571,Z 419.261,A -85,B 0,C 180,E1 -21722.497,E2 -21722.497} C_VEL
LIN {X 0,Y 215.952,Z 407.994,A -85,B 0,C 180,E1 -21724.152,E2 -21724.152} C_VEL
LIN {X 0,Y 218.764,Z 396.323,A -85,B 0,C 180,E1 -21725.47,E2 -21725.47} C_VEL
LIN {X 0,Y 221.117,Z 383.617,A -85,B 0,C 180,E1 -21726.51,E2 -21726.51} C_VEL
LIN {X 0,Y 222.885,Z 370.345,A -85,B 0,C 180,E1 -21727.213,E2 -21727.213} C_VEL
LIN {X 0,Y 224.159,Z 349.594,A -85,B 0,C 180,E1 -21727.885,E2 -21727.885} C_VEL
LIN {X 0,Y 225.619,Z 322.71,A -85,B 0,C 180,E1 -21728.676,E2 -21728.676} C_VEL
LIN {X 0,Y 224.586,Z 316.178,A -85,B 0,C 180,E1 -21729.181,E2 -21729.181} C_VEL
LIN {X 0,Y 218.698,Z 302.356,A -85,B 0,C 180,E1 -21731.183,E2 -21731.183} C_VEL
LIN {X 0,Y 213.513,Z 291.695,A -85,B 0,C 180,E1 -21733.029,E2 -21733.029} C_VEL
LIN {X 0,Y 207.19,Z 280.193,A -85,B 0,C 180,E1 -21735.425,E2 -21735.425} C_VEL
LIN {X 0,Y 203.323,Z 274.069,A -85,B 0,C 180,E1 -21736.976,E2 -21736.976} C_VEL
LIN {X 0,Y 200.713,Z 269.85,A -85,B 0,C 180,E1 -21738.091,E2 -21738.091} C_VEL
LIN {X 0,Y 197.117,Z 264.446,A -85,B 0,C 180,E1 -21739.698,E2 -21739.698} C_VEL
LIN {X 0,Y 194.13,Z 260.174,A -85,B 0,C 180,E1 -21741.114,E2 -21741.114} C_VEL
LIN {X 0,Y 193.668,Z 259.117,A -85,B 0,C 180,E1 -21741.428,E2 -21741.428} C_VEL
LIN {X 0,Y 192.552,Z 255.498,A -85,B 0,C 180,E1 -21744.59,E2 -21744.59} C_VEL
LIN {X 0,Y 192.605,Z 255.483,A -85,B 0,C 180,E1 -21747.061,E2 -21747.061} C_VEL
LIN {X 0,Y 192.622,Z 255.485,A -85,B 0,C 180,E1 -21751.685,E2 -21751.685} C_VEL
LIN {X 0,Y 192.68,Z 255.484,A -85,B 0,C 180,E1 -21756.345,E2 -21756.345} C_VEL
LIN {X 0,Y 192.7,Z 255.48,A -85,B 0,C 180,E1 -21761.487,E2 -21761.487} C_VEL
LIN {X 0,Y 192.745,Z 255.474,A -85,B 0,C 180,E1 -21765.212,E2 -21765.212} C_VEL
LIN {X 0,Y 192.982,Z 255.439,A -85,B 0,C 180,E1 -21769.509,E2 -21769.509} C_VEL
LIN {X 0,Y 193.063,Z 255.428,A -85,B 0,C 180,E1 -21771.628,E2 -21771.628} C_VEL
LIN {X 0,Y 193.259,Z 255.396,A -85,B 0,C 180,E1 -21777.916,E2 -21777.916} C_VEL
LIN {X 0,Y 193.441,Z 255.386,A -85,B 0,C 180,E1 -21780,E2 -21780} C_VEL
LIN {X 0,Y 192.963,Z 255.437,A -85,B 0,C 180,E1 -21784.178,E2 -21784.178} C_VEL
LIN {X 0,Y 193.027,Z 255.425,A -85,B 0,C 180,E1 -21788.374,E2 -21788.374} C_VEL
LIN {X 0,Y 192.796,Z 255.457,A -85,B 0,C 180,E1 -21792.634,E2 -21792.634} C_VEL
LIN {X 0,Y 192.753,Z 255.465,A -85,B 0,C 180,E1 -21796.959,E2 -21796.959} C_VEL
LIN {X 0,Y 192.636,Z 255.479,A -85,B 0,C 180,E1 -21801.398,E2 -21801.398} C_VEL
LIN {X 0,Y 192.666,Z 255.483,A -85,B 0,C 180,E1 -21804.225,E2 -21804.225} C_VEL
LIN {X 0,Y 192.652,Z 255.484,A -85,B 0,C 180,E1 -21808.892,E2 -21808.892} C_VEL
LIN {X 0,Y 192.635,Z 255.487,A -85,B 0,C 180,E1 -21812.39,E2 -21812.39} C_VEL
LIN {X 0,Y 193.458,Z 258.109,A -85,B 0,C 180,E1 -21812.911,E2 -21812.911} C_VEL
LIN {X 0,Y 195.492,Z 260.386,A -85,B 0,C 180,E1 -21813.865,E2 -21813.865} C_VEL
LIN {X 0,Y 196.471,Z 261.178,A -85,B 0,C 180,E1 -21814.291,E2 -21814.291} C_VEL
LIN {X 0,Y 198.525,Z 264.472,A -85,B 0,C 180,E1 -21815.252,E2 -21815.252} C_VEL
LIN {X 0,Y 200.305,Z 266.487,A -85,B 0,C 180,E1 -21816.006,E2 -21816.006} C_VEL
LIN {X 0,Y 203.007,Z 270.141,A -85,B 0,C 180,E1 -21817.135,E2 -21817.135} C_VEL
LIN {X 0,Y 211.67,Z 282.812,A -85,B 0,C 180,E1 -21820.458,E2 -21820.458} C_VEL
LIN {X 0,Y 216.788,Z 291.92,A -85,B 0,C 180,E1 -21822.284,E2 -21822.284} C_VEL
LIN {X 0,Y 222.871,Z 304.388,A -85,B 0,C 180,E1 -21824.348,E2 -21824.348} C_VEL
LIN {X 0,Y 226.194,Z 312.076,A -85,B 0,C 180,E1 -21825.437,E2 -21825.437} C_VEL
LIN {X 0,Y 223.503,Z 359.473,A -85,B 0,C 180,E1 -21826.867,E2 -21826.867} C_VEL
LIN {X 0,Y 222.037,Z 372.559,A -85,B 0,C 180,E1 -21827.574,E2 -21827.574} C_VEL
LIN {X 0,Y 219.866,Z 385.386,A -85,B 0,C 180,E1 -21828.603,E2 -21828.603} C_VEL
LIN {X 0,Y 217.15,Z 397.505,A -85,B 0,C 180,E1 -21829.965,E2 -21829.965} C_VEL
LIN {X 0,Y 214.228,Z 407.729,A -85,B 0,C 180,E1 -21831.441,E2 -21831.441} C_VEL
LIN {X 0,Y 210.802,Z 418.327,A -85,B 0,C 180,E1 -21833.42,E2 -21833.42} C_VEL
LIN {X 0,Y 207.588,Z 426.964,A -85,B 0,C 180,E1 -21835.453,E2 -21835.453} C_VEL
LIN {X 0,Y 204.296,Z 434.902,A -85,B 0,C 180,E1 -21837.777,E2 -21837.777} C_VEL
LIN {X 0,Y 200.908,Z 442.627,A -85,B 0,C 180,E1 -21840.677,E2 -21840.677} C_VEL
LIN {X 0,Y 197.98,Z 448.801,A -85,B 0,C 180,E1 -21843.658,E2 -21843.658} C_VEL
LIN {X 0,Y 195.494,Z 453.683,A -85,B 0,C 180,E1 -21846.706,E2 -21846.706} C_VEL
LIN {X 0,Y 193.537,Z 457.425,A -85,B 0,C 180,E1 -21849.819,E2 -21849.819} C_VEL
LIN {X 0,Y 192.043,Z 460.131,A -85,B 0,C 180,E1 -21852.976,E2 -21852.976} C_VEL
LIN {X 0,Y 191.278,Z 461.399,A -85,B 0,C 180,E1 -21855.096,E2 -21855.096} C_VEL
LIN {X 0,Y 190.664,Z 462.272,A -85,B 0,C 180,E1 -21857.223,E2 -21857.223} C_VEL
LIN {X 0,Y 190.322,Z 462.71,A -85,B 0,C 180,E1 -21859.36,E2 -21859.36} C_VEL
LIN {X 0,Y 190.177,Z 462.398,A -85,B 0,C 180,E1 -21863.635,E2 -21863.635} C_VEL
LIN {X 0,Y 190.221,Z 461.564,A -85,B 0,C 180,E1 -21866.002,E2 -21866.002} C_VEL
LIN {X 0,Y 190.524,Z 458.949,A -85,B 0,C 180,E1 -21870,E2 -21870} C_VEL
LIN {X 0,Y 191.087,Z 455.811,A -85,B 0,C 180,E1 -21873.162,E2 -21873.162} C_VEL
LIN {X 0,Y 192.005,Z 451.625,A -85,B 0,C 180,E1 -21876.304,E2 -21876.304} C_VEL
LIN {X 0,Y 193.723,Z 445.262,A -85,B 0,C 180,E1 -21879.923,E2 -21879.923} C_VEL
LIN {X 0,Y 195.634,Z 438.324,A -85,B 0,C 180,E1 -21882.975,E2 -21882.975} C_VEL
LIN {X 0,Y 198.099,Z 429.625,A -85,B 0,C 180,E1 -21885.959,E2 -21885.959} C_VEL
LIN {X 0,Y 200.451,Z 420.727,A -85,B 0,C 180,E1 -21888.394,E2 -21888.394} C_VEL
LIN {X 0,Y 202.846,Z 410.942,A -85,B 0,C 180,E1 -21890.537,E2 -21890.537} C_VEL
LIN {X 0,Y 205.11,Z 400.15,A -85,B 0,C 180,E1 -21892.408,E2 -21892.408} C_VEL
LIN {X 0,Y 207.243,Z 388.057,A -85,B 0,C 180,E1 -21894.013,E2 -21894.013} C_VEL
LIN {X 0,Y 208.961,Z 375.403,A -85,B 0,C 180,E1 -21895.26,E2 -21895.26} C_VEL
LIN {X 0,Y 210.148,Z 362.744,A -85,B 0,C 180,E1 -21896.108,E2 -21896.108} C_VEL
LIN {X 0,Y 211.14,Z 345.619,A -85,B 0,C 180,E1 -21896.747,E2 -21896.747} C_VEL
LIN {X 0,Y 213.196,Z 297.906,A -85,B 0,C 180,E1 -21898.261,E2 -21898.261} C_VEL
LIN {X 0,Y 206.941,Z 281.914,A -85,B 0,C 180,E1 -21899.988,E2 -21899.988} C_VEL
LIN {X 0,Y 202.712,Z 273.416,A -85,B 0,C 180,E1 -21901.139,E2 -21901.139} C_VEL
LIN {X 0,Y 196.411,Z 262.682,A -85,B 0,C 180,E1 -21902.892,E2 -21902.892} C_VEL
LIN {X 0,Y 194.352,Z 259.331,A -85,B 0,C 180,E1 -21903.491,E2 -21903.491} C_VEL
LIN {X 0,Y 192.914,Z 256.965,A -85,B 0,C 180,E1 -21903.921,E2 -21903.921} C_VEL
LIN {X 0,Y 192.576,Z 255.525,A -85,B 0,C 180,E1 -21904.064,E2 -21904.064} C_VEL
LIN {X 0,Y 192.553,Z 255.499,A -85,B 0,C 180,E1 -21908.351,E2 -21908.351} C_VEL
LIN {X 0,Y 192.494,Z 255.505,A -85,B 0,C 180,E1 -21913.096,E2 -21913.096} C_VEL
LIN {X 0,Y 192.494,Z 255.507,A -85,B 0,C 180,E1 -21916.904,E2 -21916.904} C_VEL
LIN {X 0,Y 192.552,Z 255.495,A -85,B 0,C 180,E1 -21921.648,E2 -21921.648} C_VEL
LIN {X 0,Y 192.598,Z 255.469,A -85,B 0,C 180,E1 -21926.814,E2 -21926.814} C_VEL
LIN {X 0,Y 192.662,Z 255.484,A -85,B 0,C 180,E1 -21931.691,E2 -21931.691} C_VEL
LIN {X 0,Y 192.707,Z 255.451,A -85,B 0,C 180,E1 -21936.348,E2 -21936.348} C_VEL
LIN {X 0,Y 192.733,Z 255.471,A -85,B 0,C 180,E1 -21941.457,E2 -21941.457} C_VEL
LIN {X 0,Y 192.765,Z 255.462,A -85,B 0,C 180,E1 -21945.214,E2 -21945.214} C_VEL
LIN {X 0,Y 192.946,Z 255.411,A -85,B 0,C 180,E1 -21949.567,E2 -21949.567} C_VEL
LIN {X 0,Y 192.975,Z 255.442,A -85,B 0,C 180,E1 -21953.727,E2 -21953.727} C_VEL
LIN {X 0,Y 193.261,Z 255.399,A -85,B 0,C 180,E1 -21957.916,E2 -21957.916} C_VEL
LIN {X 0,Y 193.441,Z 255.386,A -85,B 0,C 180,E1 -21960,E2 -21960} C_VEL
LIN {X 0,Y 192.975,Z 255.437,A -85,B 0,C 180,E1 -21964.177,E2 -21964.177} C_VEL
LIN {X 0,Y 193.08,Z 255.432,A -85,B 0,C 180,E1 -21968.372,E2 -21968.372} C_VEL
LIN {X 0,Y 193.011,Z 255.426,A -85,B 0,C 180,E1 -21970.538,E2 -21970.538} C_VEL
LIN {X 0,Y 192.72,Z 255.471,A -85,B 0,C 180,E1 -21976.962,E2 -21976.962} C_VEL
LIN {X 0,Y 192.608,Z 255.492,A -85,B 0,C 180,E1 -21981.4,E2 -21981.4} C_VEL
LIN {X 0,Y 192.64,Z 255.48,A -85,B 0,C 180,E1 -21984.208,E2 -21984.208} C_VEL
LIN {X 0,Y 192.602,Z 255.491,A -85,B 0,C 180,E1 -21988.866,E2 -21988.866} C_VEL
LIN {X 0,Y 192.595,Z 255.494,A -85,B 0,C 180,E1 -21993.187,E2 -21993.187} C_VEL
LIN {X 0,Y 192.544,Z 255.497,A -85,B 0,C 180,E1 -21998.354,E2 -21998.354} C_VEL
LIN {X 0,Y 192.487,Z 255.507,A -85,B 0,C 180,E1 -22003.094,E2 -22003.094} C_VEL
LIN {X 0,Y 192.532,Z 255.613,A -85,B 0,C 180,E1 -22007.359,E2 -22007.359} C_VEL
LIN {X 0,Y 193.873,Z 260.38,A -85,B 0,C 180,E1 -22010.096,E2 -22010.096} C_VEL
LIN {X 0,Y 201.879,Z 276.504,A -85,B 0,C 180,E1 -22012.475,E2 -22012.475} C_VEL
LIN {X 0,Y 208.721,Z 293.067,A -85,B 0,C 180,E1 -22014.428,E2 -22014.428} C_VEL
LIN {X 0,Y 209.568,Z 295.384,A -85,B 0,C 180,E1 -22014.669,E2 -22014.669} C_VEL
LIN {X 0,Y 210.407,Z 299.023,A -85,B 0,C 180,E1 -22014.958,E2 -22014.958} C_VEL
LIN {X 0,Y 210.335,Z 304.853,A -85,B 0,C 180,E1 -22015.176,E2 -22015.176} C_VEL
LIN {X 0,Y 209.26,Z 310.727,A -85,B 0,C 180,E1 -22015.226,E2 -22015.226} C_VEL
LIN {X 0,Y 206.427,Z 322.86,A -85,B 0,C 180,E1 -22015.224,E2 -22015.224} C_VEL
LIN {X 0,Y 206.011,Z 326.955,A -85,B 0,C 180,E1 -22015.317,E2 -22015.317} C_VEL
LIN {X 0,Y 203.978,Z 369.777,A -85,B 0,C 180,E1 -22016.767,E2 -22016.767} C_VEL
LIN {X 0,Y 202.612,Z 382.781,A -85,B 0,C 180,E1 -22017.55,E2 -22017.55} C_VEL
LIN {X 0,Y 200.852,Z 394.82,A -85,B 0,C 180,E1 -22018.635,E2 -22018.635} C_VEL
LIN {X 0,Y 198.736,Z 406.175,A -85,B 0,C 180,E1 -22020.033,E2 -22020.033} C_VEL
LIN {X 0,Y 196.097,Z 417.883,A -85,B 0,C 180,E1 -22021.94,E2 -22021.94} C_VEL
LIN {X 0,Y 193.343,Z 428.402,A -85,B 0,C 180,E1 -22024.138,E2 -22024.138} C_VEL
LIN {X 0,Y 190.926,Z 437.694,A -85,B 0,C 180,E1 -22026.625,E2 -22026.625} C_VEL
LIN {X 0,Y 188.432,Z 447.018,A -85,B 0,C 180,E1 -22029.818,E2 -22029.818} C_VEL
LIN {X 0,Y 186.317,Z 454.363,A -85,B 0,C 180,E1 -22033.002,E2 -22033.002} C_VEL
LIN {X 0,Y 184.944,Z 459.33,A -85,B 0,C 180,E1 -22035.7,E2 -22035.7} C_VEL
LIN {X 0,Y 183.933,Z 464.157,A -85,B 0,C 180,E1 -22038.986,E2 -22038.986} C_VEL
LIN {X 0,Y 183.316,Z 467.848,A -85,B 0,C 180,E1 -22042.289,E2 -22042.289} C_VEL
LIN {X 0,Y 183.074,Z 471.084,A -85,B 0,C 180,E1 -22046.477,E2 -22046.477} C_VEL
LIN {X 0,Y 183.186,Z 472.607,A -85,B 0,C 180,E1 -22050,E2 -22050} C_VEL
LIN {X 0,Y 183.053,Z 473.079,A -85,B 0,C 180,E1 -22053.414,E2 -22053.414} C_VEL
LIN {X 0,Y 183.213,Z 472.639,A -85,B 0,C 180,E1 -22056.608,E2 -22056.608} C_VEL
LIN {X 0,Y 183.518,Z 471.88,A -85,B 0,C 180,E1 -22058.812,E2 -22058.812} C_VEL
LIN {X 0,Y 184.063,Z 470.686,A -85,B 0,C 180,E1 -22061.006,E2 -22061.006} C_VEL
LIN {X 0,Y 185.255,Z 468.149,A -85,B 0,C 180,E1 -22064.276,E2 -22064.276} C_VEL
LIN {X 0,Y 187.063,Z 464.619,A -85,B 0,C 180,E1 -22067.491,E2 -22067.491} C_VEL
LIN {X 0,Y 189.498,Z 460.004,A -85,B 0,C 180,E1 -22070.63,E2 -22070.63} C_VEL
LIN {X 0,Y 193.023,Z 452.871,A -85,B 0,C 180,E1 -22074.271,E2 -22074.271} C_VEL
LIN {X 0,Y 196.326,Z 445.536,A -85,B 0,C 180,E1 -22077.156,E2 -22077.156} C_VEL
LIN {X 0,Y 199.701,Z 437.882,A -85,B 0,C 180,E1 -22079.518,E2 -22079.518} C_VEL
